	            "Cip".obiekt[#nr].inStartAuto := "Cip".obiekt["Cip".tor[2].pompkaDozowaniaDezynfekantuwLinię].outStartUrządzenie;
	      
	        0:
	            "Cip".obiekt[#nr].Flipaj.in := 0;
	    END_CASE;
	END_REGION
	    
	    REGION ZAWOR ZRZUTOWY DO KANALIZACJI
	    
	    
	        #nr := "Cip".tor[2].zawórZrzutowyDoKanalizacji;
	    CASE "Tor2_program".program.numerKroku OF
	    7100, 7202..7246, 7270,7287,7310, 7320, 7321, 7402, 7403, 7411..7414, 7420, 7431..7435, 7440, 7460:
	    "Cip".obiekt[#nr].procedura := 2;
	   
	    ELSE
	    "Cip".obiekt[#nr].procedura := 0;
	    
	    END_CASE;
	    
	    CASE "Cip".obiekt[#nr].procedura OF
	    2:
	    //wyzwolenie timerków
	    "Cip".obiekt[#nr].SetReset.czasDoSet := 2;
	    "Cip".obiekt[#nr].SetReset.inSet :=
	    "Cip".obiekt["Cip".tor[2].zawórPowrotnyWodyWtórnej].outStartUrządzenie
	    OR "Cip".obiekt["Cip".tor[2].zawórPowrotnyŁugu].outStartUrządzenie
	    OR "Cip".obiekt["Cip".tor[2].zawórPowrotnyKwasu].outStartUrządzenie;
	    
	    "Cip".obiekt[#nr].SetReset.czasDoReset := 2;
	    "Cip".obiekt[#nr].SetReset.inReset :=
	    NOT "Cip".obiekt["Cip".tor[2].zawórPowrotnyWodyWtórnej].outStartUrządzenie
	    AND NOT "Cip".obiekt["Cip".tor[2].zawórPowrotnyŁugu].outStartUrządzenie
	    AND NOT "Cip".obiekt["Cip".tor[2].zawórPowrotnyKwasu].outStartUrządzenie;
	    //załaczanie
	    "Cip".obiekt[#nr].inStartAuto := "Cip".obiekt[#nr].SetReset.wyjście;
	    
	    3:
	    //wyzwolenie timerków
	    "Cip".obiekt[#nr].SetReset.czasDoSet := 2;
	    "Cip".obiekt[#nr].SetReset.inSet :=
	    "Cip".obiekt["Cip".tor[2].zawórBypassPrzygotowaniaStacji].outStartUrządzenie;
	    
	    
	    "Cip".obiekt[#nr].SetReset.czasDoReset := 2;
	    "Cip".obiekt[#nr].SetReset.inReset :=
	    NOT "Cip".obiekt["Cip".tor[2].zawórBypassPrzygotowaniaStacji].outStartUrządzenie;
	    
	    //załaczanie
	    "Cip".obiekt[#nr].inStartAuto := "Cip".obiekt[#nr].SetReset.wyjście;
	    END_CASE;
	    END_REGION
	    
	    REGION ZAWOR WYDAWCZY CIP
	    
	        #nr := "Cip".tor[2].zawórWydawczyCip;
	    CASE "Tor2_program".program.numerKroku OF
	    7210..7290:
	    "Cip".obiekt[#nr].procedura := 1;
	    
	    ELSE
	    "Cip".obiekt[#nr].procedura := 0;
	    
	    END_CASE;
	    
	    CASE "Cip".obiekt[#nr].procedura OF
	    2:
	    //wyzwolenie timerków
	    "Cip".obiekt[#nr].SetReset.czasDoSet := 2;
	    "Cip".obiekt[#nr].SetReset.inSet :=
	    "Cip".obiekt["Cip".tor[2].pompaPodawaniaCip].outStartUrządzenie;
	    
	    "Cip".obiekt[#nr].SetReset.czasDoReset := 2;
	    "Cip".obiekt[#nr].SetReset.inReset :=
	    NOT "Cip".obiekt["Cip".tor[2].pompaPodawaniaCip].outStartUrządzenie;
	    //załaczanie
	    "Cip".obiekt[#nr].inStartAuto := "Cip".obiekt[#nr].SetReset.wyjście;
	    
	    END_CASE;
	    END_REGION
	    
	    REGION ZAWOR BYPASS PRZYGOTOWANIA STACJI
	    
	        #nr := "Cip".tor[2].zawórBypassPrzygotowaniaStacji;
	    CASE "Tor2_program".program.numerKroku OF
	    7210..7290:
	    "Cip".obiekt[#nr].procedura := 2;
	    7320:
	    "Cip".obiekt[#nr].procedura := 3;
	    ELSE
	    "Cip".obiekt[#nr].procedura := 0;
	    
	    END_CASE;
	    CASE "Cip".obiekt[#nr].procedura OF
	    2:
	    //wyzwolenie timerków
	    "Cip".obiekt[#nr].SetReset.czasDoSet := 2;
	    "Cip".obiekt[#nr].SetReset.inSet :=NOT 
	    "Cip".obiekt["Cip".tor[2].zawórWydawczyCip].outStartUrządzenie;
	    
	    "Cip".obiekt[#nr].SetReset.czasDoReset := 2;
	    "Cip".obiekt[#nr].SetReset.inReset :=
	    "Cip".obiekt["Cip".tor[2].zawórWydawczyCip].outStartUrządzenie;
	    //załaczanie
	    "Cip".obiekt[#nr].inStartAuto := "Cip".obiekt[#nr].SetReset.wyjście;
	    3:
	    
	    //załaczanie
	    "Cip".obiekt[#nr].inStartAuto := 1;
	    
	    END_CASE;
	    END_REGION
	    
	    REGION ZAWOR WYDAWCZY WODY WTORNEJ
	    
	        #nr := "Cip".tor[2].zawórWydawczyWodyWtórnej;
	    
	    CASE "Tor2_program".program.numerKroku OF
	    7210,7230:
	    "Cip".obiekt[#nr].procedura := 2;
	    7100:
	    "Cip".obiekt[#nr].procedura := 3;
	    ELSE
	    "Cip".obiekt[#nr].procedura := 0;
	    
	    END_CASE;
	    
	    
	    
	    CASE "Cip".obiekt[#nr].procedura OF
	    2:
	    //wyzwolenie timerków
	    "Cip".obiekt[#nr].SetReset.czasDoSet := 3;
	    "Cip".obiekt[#nr].SetReset.inSet :=
	    "Cip".obiekt["Cip".tor[0].zbiornikWodyWtórnej.czujnikDolnegoPoziomu].hmiPotwWysterowania
	    AND (#aktualnyKrokMycia = 1 OR #aktualnyKrokMycia = 2);
	    
	    "Cip".obiekt[#nr].SetReset.czasDoReset := 10;
	    "Cip".obiekt[#nr].SetReset.inReset :=
	    NOT "Cip".obiekt["Cip".tor[0].zbiornikWodyWtórnej.czujnikDolnegoPoziomu].hmiPotwWysterowania
	    OR (#aktualnyKrokMycia <> 1 AND #aktualnyKrokMycia <> 2);
	    //załaczanie
	    "Cip".obiekt[#nr].inStartAuto := "Cip".obiekt[#nr].SetReset.wyjście;
	    3:
	    //wyzwolenie timerków
	    "Cip".obiekt[#nr].SetReset.czasDoSet := 3;
	    "Cip".obiekt[#nr].SetReset.inSet :=
	    ("Tor2_program".program.numerKroku >= 7401 AND
	    "Tor2_program".program.numerKroku <= 7420);
	    
	    
	    "Cip".obiekt[#nr].SetReset.czasDoReset := 60;
	    "Cip".obiekt[#nr].SetReset.inReset :=
	    NOT ("Tor2_program".program.numerKroku >= 7401 AND
	    "Tor2_program".program.numerKroku <= 7420);
	    
	    //załaczanie
	    "Cip".obiekt[#nr].inStartAuto := "Cip".obiekt[#nr].SetReset.wyjście;
	    
	    END_CASE;
	    END_REGION
	    
	    REGION ZAWÓR POWROTNY WODY WTORNEJ
	    
	        #nr := "Cip".tor[2].zawórPowrotnyWodyWtórnej;
	    CASE "Tor2_program".program.numerKroku OF
	        7250, 7270, 7285, 7287:
	            "Cip".obiekt[#nr].procedura := 2;
	        7402, 7403, 7411, 7414, 7420:
	            "Cip".obiekt[#nr].procedura := 1;
	        ELSE
	            "Cip".obiekt[#nr].procedura := 0;
	            
	    END_CASE;
	    
	    CASE "Cip".obiekt[#nr].procedura OF
	    2:
	    //wyzwolenie timerków
	    "Cip".obiekt[#nr].SetReset.czasDoSet := 1;
	    "Cip".obiekt[#nr].SetReset.inSet :=
	    NOT "Cip".obiekt["Cip".tor[0].zbiornikWodyWtórnej.czujnikGórnegoPoziomu].hmiPotwWysterowania
	    // AND (#aktualnyKrokMycia = 5 OR #aktualnyKrokMycia = 6); // nie wiem czy to było dobrze w Orle 1
	    ;
	    "Cip".obiekt[#nr].SetReset.czasDoReset := 1;
	    "Cip".obiekt[#nr].SetReset.inReset :=
	    "Cip".obiekt["Cip".tor[0].zbiornikWodyWtórnej.czujnikGórnegoPoziomu].hmiPotwWysterowania
	    // OR (#aktualnyKrokMycia <> 5 AND #aktualnyKrokMycia <> 6);
	     ;
	    // ;
	    //załaczanie
	    "Cip".obiekt[#nr].inStartAuto := "Cip".obiekt[#nr].SetReset.wyjście;
	    
	    
	    END_CASE;
	    END_REGION
	    
	    REGION ZAWOR WYDAWCZY ŁUGU
	    
	        #nr := "Cip".tor[2].zawórWydawczyŁugu;
	        CASE "Tor2_program".program.numerKroku OF
	            7240..7243,7411,7412:
	                "Cip".obiekt[#nr].procedura := 2;
	            7100:
	                "Cip".obiekt[#nr].procedura := 3;
	            7320:
	                "Cip".obiekt[#nr].procedura := 4;
	            ELSE
	                "Cip".obiekt[#nr].procedura := 0;
	                
	        END_CASE;
	        
	    CASE "Cip".obiekt[#nr].procedura OF
	    2:
	    //wyzwolenie timerków
	    "Cip".obiekt[#nr].SetReset.czasDoSet := 3;
	    "Cip".obiekt[#nr].SetReset.inSet :=
	    "Cip".obiekt["Cip".tor[0].zbiornikŁugu.czujnikDolnegoPoziomu].hmiPotwWysterowania
	    AND (#aktualnyKrokMycia = 3);
	    
	    "Cip".obiekt[#nr].SetReset.czasDoReset := 10;
	    "Cip".obiekt[#nr].SetReset.inReset :=
	    NOT "Cip".obiekt["Cip".tor[0].zbiornikŁugu.czujnikDolnegoPoziomu].hmiPotwWysterowania
	    OR (#aktualnyKrokMycia <> 3);
	    //załaczanie
	    "Cip".obiekt[#nr].inStartAuto := "Cip".obiekt[#nr].SetReset.wyjście;
	    3:
	    //wyzwolenie timerków
	    "Cip".obiekt[#nr].SetReset.czasDoSet := 3;
	    "Cip".obiekt[#nr].SetReset.inSet :=
	    ("Tor2_program".program.numerKroku >= 7430 AND
	    "Tor2_program".program.numerKroku <= 7440);
	    
	    
	    "Cip".obiekt[#nr].SetReset.czasDoReset := 3;
	    "Cip".obiekt[#nr].SetReset.inReset :=
	    NOT ("Tor2_program".program.numerKroku >= 7430 AND
	    "Tor2_program".program.numerKroku <= 7440);
	    
	    //załaczanie
	    "Cip".obiekt[#nr].inStartAuto := "Cip".obiekt[#nr].SetReset.wyjście;
	    
	    4:
	    //wyzwolenie timerków
	    "Cip".obiekt[#nr].SetReset.czasDoSet := 3;
	    "Cip".obiekt[#nr].SetReset.inSet :=
	    "Cip".obiekt["Cip".tor[0].zbiornikŁugu.czujnikGórnegoPoziomu].hmiPotwWysterowania
	    AND (#aktualnyKrokMycia = 3);
	    
	    
	    
	    "Cip".obiekt[#nr].SetReset.czasDoReset := 3;
	    "Cip".obiekt[#nr].SetReset.inReset :=
	    NOT "Cip".obiekt["Cip".tor[0].zbiornikŁugu.czujnikGórnegoPoziomu].hmiPotwWysterowania
	    OR (#aktualnyKrokMycia <> 3);
	    
	    //załaczanie
	    "Cip".obiekt[#nr].inStartAuto := "Cip".obiekt[#nr].SetReset.wyjście;
	    
	    
	    
	    
	    
	    
	    
	    
	    END_CASE;
	    END_REGION
	    
	    REGION ZAWÓR POWROTNY ŁUGU
	    
	        #nr := "Cip".tor[2].zawórPowrotnyŁugu;
	        CASE "Tor2_program".program.numerKroku OF
	            7431,7432,7434,7435,7440:
	                "Cip".obiekt[#nr].procedura := 1;
	            7242, 7245, 7246, 7321:
	                "Cip".obiekt[#nr].procedura := 2;
	            7100:
	                "Cip".obiekt[#nr].procedura := 3;
	            7243, 7244, 7310, 7320:
	                "Cip".obiekt[#nr].procedura := 4;
	            ELSE
	                "Cip".obiekt[#nr].procedura := 0;
	        END_CASE;
	        
	    CASE "Cip".obiekt[#nr].procedura OF
	    2:
	    //wyzwolenie timerków
	    "Cip".obiekt[#nr].SetReset.czasDoSet := 1;
	    "Cip".obiekt[#nr].SetReset.inSet :=
	    "Cip".obiekt["Cip".tor[2].przewodnośćNaPowrocie].WartośćPomiaru >=
	    "Tor2_RecepturyStacjaMycia".Receptura[#aktualnyNumerReceptury].Krok[#aktualnyKrokMycia].PM[10]
	    AND (#aktualnyKrokMycia = 3)
	    AND NOT "Cip".obiekt["Cip".tor[0].zbiornikŁugu.czujnikGórnegoPoziomu].hmiPotwWysterowania;
	    
	    "Cip".obiekt[#nr].SetReset.czasDoReset := 1;
	    "Cip".obiekt[#nr].SetReset.inReset :=
	    "Cip".obiekt["Cip".tor[2].przewodnośćNaPowrocie].WartośćPomiaru <
	    "Tor2_RecepturyStacjaMycia".Receptura[#aktualnyNumerReceptury].Krok[#aktualnyKrokMycia].PM[10]
	    OR (#aktualnyKrokMycia <> 3)
	    OR "Cip".obiekt["Cip".tor[0].zbiornikŁugu.czujnikGórnegoPoziomu].hmiPotwWysterowania;
	    //załaczanie
	    "Cip".obiekt[#nr].inStartAuto := "Cip".obiekt[#nr].SetReset.wyjście;
	    3:
	    //wyzwolenie timerków
	    "Cip".obiekt[#nr].SetReset.czasDoSet := 3;
	    "Cip".obiekt[#nr].SetReset.inSet :=
	    "Cip".obiekt["Cip".tor[2].zawórWydawczyŁugu].inStartAuto
	    AND ("Tor2_program".program.numerKroku > 7400
	    AND "Tor2_program".program.numerKroku < 7470);
	    
	    
	    "Cip".obiekt[#nr].SetReset.czasDoReset := 3;
	    "Cip".obiekt[#nr].SetReset.inReset :=
	    NOT "Cip".obiekt["Cip".tor[2].zawórWydawczyŁugu].inStartAuto
	    OR ("Tor2_program".program.numerKroku < 7400
	    OR "Tor2_program".program.numerKroku > 7470);
	    
	    //załaczanie
	    "Cip".obiekt[#nr].inStartAuto := "Cip".obiekt[#nr].SetReset.wyjście;
	    
	    4:
	    //wyzwolenie timerków
	    "Cip".obiekt[#nr].SetReset.czasDoSet := 3;
	    "Cip".obiekt[#nr].SetReset.inSet :=
	    (#aktualnyKrokMycia = 3);
	    
	    "Cip".obiekt[#nr].SetReset.czasDoReset := 10;
	    "Cip".obiekt[#nr].SetReset.inReset :=
	    (#aktualnyKrokMycia <> 3);
	    //załaczanie
	    "Cip".obiekt[#nr].inStartAuto := "Cip".obiekt[#nr].SetReset.wyjście;
	    END_CASE;
	    
	    END_REGION
	    
	    REGION ZAWÓR WYDAWCZY KWASU
	        
	        #nr := "Cip".tor[2].zawórWydawczyKwasu;
	        CASE "Tor2_program".program.numerKroku OF
	            7240..7243, 7411, 7412, 7434, 7435:
	                "Cip".obiekt[#nr].procedura := 2;
	            7100:
	                "Cip".obiekt[#nr].procedura := 3;
	            7320:
	                "Cip".obiekt[#nr].procedura := 4;
	            ELSE
	                "Cip".obiekt[#nr].procedura := 0;
	                
	        END_CASE;
	        
	        CASE "Cip".obiekt[#nr].procedura OF
	            2:
	                //wyzwolenie timerków
	                "Cip".obiekt[#nr].SetReset.czasDoSet := 3;
	                "Cip".obiekt[#nr].SetReset.inSet :=
	                "Cip".obiekt["Cip".tor[0].zbiornikKwasu.czujnikDolnegoPoziomu].hmiPotwWysterowania
	                AND (#aktualnyKrokMycia = 4);
	                
	                "Cip".obiekt[#nr].SetReset.czasDoReset := 10;
	                "Cip".obiekt[#nr].SetReset.inReset :=
	                NOT "Cip".obiekt["Cip".tor[0].zbiornikKwasu.czujnikDolnegoPoziomu].hmiPotwWysterowania
	                OR (#aktualnyKrokMycia <> 4);
	                
	                //załaczanie
	                "Cip".obiekt[#nr].inStartAuto := "Cip".obiekt[#nr].SetReset.wyjście;
	            3:
	                //wyzwolenie timerków
	                "Cip".obiekt[#nr].SetReset.czasDoSet := 3;
	                "Cip".obiekt[#nr].SetReset.inSet :=
	                ("Tor2_program".program.numerKroku >= 7450 AND
	                "Tor2_program".program.numerKroku <= 7470);
	                
	                
	                "Cip".obiekt[#nr].SetReset.czasDoReset := 3;
	                "Cip".obiekt[#nr].SetReset.inReset :=
	                NOT ("Tor2_program".program.numerKroku >= 7450 AND
	                "Tor2_program".program.numerKroku <= 7470);
	                
	                //załaczanie
	                "Cip".obiekt[#nr].inStartAuto := "Cip".obiekt[#nr].SetReset.wyjście;
	                
	                
	            4:
	                //wyzwolenie timerków
	                "Cip".obiekt[#nr].SetReset.czasDoSet := 3;
	                "Cip".obiekt[#nr].SetReset.inSet :=
	                "Cip".obiekt["Cip".tor[0].zbiornikKwasu.czujnikGórnegoPoziomu].hmiPotwWysterowania
	                AND (#aktualnyKrokMycia = 4);
	                
	                
	                
	                "Cip".obiekt[#nr].SetReset.czasDoReset := 3;
	                "Cip".obiekt[#nr].SetReset.inReset :=
	                NOT "Cip".obiekt["Cip".tor[0].zbiornikKwasu.czujnikGórnegoPoziomu].hmiPotwWysterowania
	                OR (#aktualnyKrokMycia <> 4);
	                
	                //załaczanie
	                "Cip".obiekt[#nr].inStartAuto := "Cip".obiekt[#nr].SetReset.wyjście;
	                
	        END_CASE;
	    END_REGION
	    
	    REGION ZAWÓR POWROTNY KWASU
	        
	        #nr := "Cip".tor[2].zawórPowrotnyKwasu;
	        
	        CASE "Tor2_program".program.numerKroku OF
	            7460:
	                "Cip".obiekt[#nr].procedura := 1;
	            7242, 7245, 7246, 7321:
	                "Cip".obiekt[#nr].procedura := 2;
	            7100:
	                "Cip".obiekt[#nr].procedura := 3;
	            7243, 7244, 7310, 7320:
	                "Cip".obiekt[#nr].procedura := 4;
	            ELSE
	                "Cip".obiekt[#nr].procedura := 0;
	        END_CASE;
	        
	        CASE "Cip".obiekt[#nr].procedura OF
	            2:
	                //wyzwolenie timerków
	                "Cip".obiekt[#nr].SetReset.czasDoSet := 1;
	                "Cip".obiekt[#nr].SetReset.inSet :=
	                "Cip".obiekt["Cip".tor[2].przewodnośćNaPowrocie].WartośćPomiaru >=
	                "Tor2_RecepturyStacjaMycia".Receptura[#aktualnyNumerReceptury].Krok[#aktualnyKrokMycia].PM[10]
	                AND (#aktualnyKrokMycia = 4)
	                AND NOT "Cip".obiekt["Cip".tor[0].zbiornikKwasu.czujnikGórnegoPoziomu].hmiPotwWysterowania;
	                
	                "Cip".obiekt[#nr].SetReset.czasDoReset := 1;
	                "Cip".obiekt[#nr].SetReset.inReset :=
	                "Cip".obiekt["Cip".tor[2].przewodnośćNaPowrocie].WartośćPomiaru <
	                "Tor2_RecepturyStacjaMycia".Receptura[#aktualnyNumerReceptury].Krok[#aktualnyKrokMycia].PM[10]
	                OR (#aktualnyKrokMycia <> 4)
	                OR "Cip".obiekt["Cip".tor[0].zbiornikKwasu.czujnikGórnegoPoziomu].hmiPotwWysterowania;
	                //załaczanie
	                "Cip".obiekt[#nr].inStartAuto := "Cip".obiekt[#nr].SetReset.wyjście;
	            3:
	                //wyzwolenie timerków
	                "Cip".obiekt[#nr].SetReset.czasDoSet := 3;
	                "Cip".obiekt[#nr].SetReset.inSet :=
	                "Cip".obiekt["Cip".tor[2].zawórWydawczyKwasu].inStartAuto AND
	                ("Tor2_program".program.numerKroku >= 7400 AND
	                "Tor2_program".program.numerKroku <= 7470);
	                ;
	                
	                
	                "Cip".obiekt[#nr].SetReset.czasDoReset := 3;
	                "Cip".obiekt[#nr].SetReset.inReset :=
	                NOT "Cip".obiekt["Cip".tor[2].zawórWydawczyKwasu].inStartAuto
	                OR ("Tor2_program".program.numerKroku < 7400 OR
	                "Tor2_program".program.numerKroku > 7470);
	                ;
	                
	                //załaczanie
	                "Cip".obiekt[#nr].inStartAuto := "Cip".obiekt[#nr].SetReset.wyjście;
	            4:
	                //wyzwolenie timerków
	                "Cip".obiekt[#nr].SetReset.czasDoSet := 3;
	                "Cip".obiekt[#nr].SetReset.inSet := (#aktualnyKrokMycia = 4);
	                
	                "Cip".obiekt[#nr].SetReset.czasDoReset := 10;
	                "Cip".obiekt[#nr].SetReset.inReset := (#aktualnyKrokMycia <> 4);
	                
	                //załaczanie
	                "Cip".obiekt[#nr].inStartAuto := "Cip".obiekt[#nr].SetReset.wyjście;
	        END_CASE;
	    END_REGION
	    
	    REGION ZAWÓR WYDAWCZY WODY CZYSTEJ
	    
	        #nr := "Cip".tor[2].zawórWydawczyWodyCzystej;
	        
	        CASE "Tor2_program".program.numerKroku OF
	            7220..7230, 7411, 7412:
	                "Cip".obiekt[#nr].procedura := 2;
	            7244..7270, 7321, 7402, 7403, 7414, 7420, 7431, 7432, 7440, 7460:
	                "Cip".obiekt[#nr].procedura := 3;
	            7242, 7243:
	                "Cip".obiekt[#nr].procedura := 4;
	            7310, 7320:
	                "Cip".obiekt[#nr].procedura := 5;
	            7281..7291:
	                "Cip".obiekt[#nr].procedura := 6;
	            ELSE
	                "Cip".obiekt[#nr].procedura := 0;
	                
	        END_CASE;
	        
	        
	    CASE "Cip".obiekt[#nr].procedura OF
	    2:
	    //wyzwolenie timerków
	    "Cip".obiekt[#nr].SetReset.czasDoSet := 3;
	    "Cip".obiekt[#nr].SetReset.inSet :=
	    "Cip".obiekt["Cip".tor[0].zbiornikwodyCzystej.czujnikDolnegoPoziomu].hmiPotwWysterowania
	    AND NOT "Cip".obiekt["Cip".tor[0].zbiornikWodyWtórnej.czujnikDolnegoPoziomu].hmiPotwWysterowania;
	    
	    "Cip".obiekt[#nr].SetReset.czasDoReset := 10;
	    "Cip".obiekt[#nr].SetReset.inReset :=
	    NOT "Cip".obiekt["Cip".tor[0].zbiornikwodyCzystej.czujnikDolnegoPoziomu].hmiPotwWysterowania
	    OR "Cip".obiekt["Cip".tor[0].zbiornikWodyWtórnej.czujnikDolnegoPoziomu].hmiPotwWysterowania;
	    //załaczanie
	    "Cip".obiekt[#nr].inStartAuto := "Cip".obiekt[#nr].SetReset.wyjście;
	    3:
	    //wyzwolenie timerków
	    "Cip".obiekt[#nr].SetReset.czasDoSet := 3;
	    "Cip".obiekt[#nr].SetReset.inSet :=
	    "Cip".obiekt["Cip".tor[0].zbiornikwodyCzystej.czujnikDolnegoPoziomu].hmiPotwWysterowania;
	    
	    
	    "Cip".obiekt[#nr].SetReset.czasDoReset := 3;
	    "Cip".obiekt[#nr].SetReset.inReset :=
	    NOT "Cip".obiekt["Cip".tor[0].zbiornikwodyCzystej.czujnikDolnegoPoziomu].hmiPotwWysterowania;
	    
	    //załaczanie
	    "Cip".obiekt[#nr].inStartAuto := "Cip".obiekt[#nr].SetReset.wyjście;
	    
	    4:
	    //wyzwolenie timerków
	    "Cip".obiekt[#nr].SetReset.czasDoSet := 1;
	    "Cip".obiekt[#nr].SetReset.inSet :=
	    (NOT "Cip".obiekt["Cip".tor[0].zbiornikŁugu.czujnikDolnegoPoziomu].hmiPotwWysterowania AND #aktualnyKrokMycia = 3)
	    OR (NOT "Cip".obiekt["Cip".tor[0].zbiornikKwasu.czujnikDolnegoPoziomu].hmiPotwWysterowania AND #aktualnyKrokMycia = 4);
	    
	    
	    "Cip".obiekt[#nr].SetReset.czasDoReset := 5;
	    "Cip".obiekt[#nr].SetReset.inReset :=
	    ("Cip".obiekt["Cip".tor[0].zbiornikŁugu.czujnikDolnegoPoziomu].hmiPotwWysterowania AND #aktualnyKrokMycia = 3)
	    OR ("Cip".obiekt["Cip".tor[0].zbiornikKwasu.czujnikDolnegoPoziomu].hmiPotwWysterowania AND #aktualnyKrokMycia = 4);
	    //załaczanie
	    "Cip".obiekt[#nr].inStartAuto := "Cip".obiekt[#nr].SetReset.wyjście;
	    
	    5:
	    //wyzwolenie timerków
	    "Cip".obiekt[#nr].SetReset.czasDoSet := 1;
	    "Cip".obiekt[#nr].SetReset.inSet :=
	    (NOT "Cip".obiekt["Cip".tor[0].zbiornikŁugu.czujnikGórnegoPoziomu].hmiPotwWysterowania AND #aktualnyKrokMycia = 3)
	    OR (NOT "Cip".obiekt["Cip".tor[0].zbiornikKwasu.czujnikGórnegoPoziomu].hmiPotwWysterowania AND #aktualnyKrokMycia = 4);
	    
	    
	    "Cip".obiekt[#nr].SetReset.czasDoReset := 2;
	    "Cip".obiekt[#nr].SetReset.inReset :=
	    ("Cip".obiekt["Cip".tor[0].zbiornikŁugu.czujnikGórnegoPoziomu].hmiPotwWysterowania AND #aktualnyKrokMycia = 3)
	    OR ("Cip".obiekt["Cip".tor[0].zbiornikKwasu.czujnikGórnegoPoziomu].hmiPotwWysterowania AND #aktualnyKrokMycia = 4);
	    //załaczanie
	    "Cip".obiekt[#nr].inStartAuto := "Cip".obiekt[#nr].SetReset.wyjście;
	6:
	    //wyzwolenie timerków
	    "Cip".obiekt[#nr].SetReset.czasDoSet :=1;
	    "Cip".obiekt[#nr].SetReset.inSet :=
	    NOT ("Cip".obiekt["Cip".tor[2].zawórWydawczyDezynfekantu].hmiPotwWysterowania);
	    
	    
	    "Cip".obiekt[#nr].SetReset.czasDoReset := 2;
	    "Cip".obiekt[#nr].SetReset.inReset :=
	    ("Cip".obiekt["Cip".tor[2].zawórWydawczyDezynfekantu].hmiPotwWysterowania);;
	    //załaczanie
	    "Cip".obiekt[#nr].inStartAuto := "Cip".obiekt[#nr].SetReset.wyjście;
	    
	    END_CASE;
	    END_REGION
	    
	    REGION zawór wydawczy dezynfekantu
	        
	        #nr := "Cip".tor[2].zawórWydawczyDezynfekantu;
	        CASE "Tor2_program".program.numerKroku OF
	            7282..7284:
	                "Cip".obiekt[#nr].procedura := 2;
	                
	            ELSE
	                "Cip".obiekt[#nr].procedura := 0;
	                
	        END_CASE;
	        
	        CASE "Cip".obiekt[#nr].procedura OF
	            2:
	                //wyzwolenie timerków
	                "Cip".obiekt[#nr].SetReset.czasDoSet := 2;
	                "Cip".obiekt[#nr].SetReset.inSet :=
	                "Cip".obiekt["Cip".tor[2].zbiornikDezynfekantu.poziomAnalogowy].WartośćPomiaru > 10.0;
	                
	                "Cip".obiekt[#nr].SetReset.czasDoReset := 2;
	                "Cip".obiekt[#nr].SetReset.inReset :=
	                "Cip".obiekt["Cip".tor[2].zbiornikDezynfekantu.poziomAnalogowy].WartośćPomiaru < 0.01;
	                ;
	                //załaczanie
	                "Cip".obiekt[#nr].inStartAuto := "Cip".obiekt[#nr].SetReset.wyjście;
	                
	        END_CASE;
	    END_REGION
	    
	    REGION zawór powrotny dezynfekantu
	        
	        #nr := "Cip".tor[2].zawórPowrotnyDezynfekantu;
	        CASE "Tor2_program".program.numerKroku OF
	            7281..7283:
	                "Cip".obiekt[#nr].procedura :=2;
	                
	            ELSE
	                "Cip".obiekt[#nr].procedura := 0;
	                
	        END_CASE;
	        
	        CASE "Cip".obiekt[#nr].procedura OF
	            2:
	                //wyzwolenie timerków
	                "Cip".obiekt[#nr].SetReset.czasDoSet := 5;
	                "Cip".obiekt[#nr].SetReset.inSet :=
	                NOT  "Cip".obiekt["Cip".tor[2].zbiornikDezynfekantu.czujnikGórnegoPoziomu].hmiPotwWysterowania ;
	                
	                "Cip".obiekt[#nr].SetReset.czasDoReset := 0;
	                "Cip".obiekt[#nr].SetReset.inReset :=
	                "Cip".obiekt["Cip".tor[2].zbiornikDezynfekantu.czujnikGórnegoPoziomu].hmiPotwWysterowania;
	                ;
	                //załaczanie
	                "Cip".obiekt[#nr].inStartAuto := "Cip".obiekt[#nr].SetReset.wyjście;
	                
	        END_CASE;
	    END_REGION
	    
	    REGION zawór stopowy dezynfekantu
	        
	        #nr := "Cip".tor[2].zawórStopowyPowrotuDezynfekantu;
	        CASE "Tor2_program".program.numerKroku OF
	            7281..7283:
	                "Cip".obiekt[#nr].procedura := 2;
	                
	            ELSE
	                "Cip".obiekt[#nr].procedura := 0;
	                
	        END_CASE;
	        
	        CASE "Cip".obiekt[#nr].procedura OF
	            2:
	                //wyzwolenie timerków
	                "Cip".obiekt[#nr].SetReset.czasDoSet := 0;
	                "Cip".obiekt[#nr].SetReset.inSet :=
	                "Cip".obiekt["Cip".tor[2].zawórPowrotnyDezynfekantu].hmiPotwWysterowania;
	                
	                "Cip".obiekt[#nr].SetReset.czasDoReset := 0;
	                "Cip".obiekt[#nr].SetReset.inReset :=
	                NOT "Cip".obiekt["Cip".tor[2].zawórPowrotnyDezynfekantu].hmiPotwWysterowania;
	                ;
	                //załaczanie
	                "Cip".obiekt[#nr].inStartAuto := "Cip".obiekt[#nr].SetReset.wyjście;
	                
	        END_CASE;
	    END_REGION
	    
	    REGION ZAWÓR PAROWY REGULACYJNY
	    
	        #nr := "Cip".tor[2].zawórParowyRegulacyjny;
	        
	    CASE "Tor2_program".program.numerKroku OF
	    7220, 7250, 7403, 7414, 7432:
	    "Cip".obiekt[#nr].procedura := 2;
	    7242..7246, 7320, 7321, 7411, 7412, 7434, 7435:
	    "Cip".obiekt[#nr].procedura := 3;
	    
	    ELSE
	    "Cip".obiekt[#nr].procedura := 0;
	    
	    END_CASE;
	    
	    
	    CASE "Cip".obiekt[#nr].procedura OF
	    2:
	    //wyzwolenie timerków
	    "Cip".obiekt[#nr].SetReset.czasDoSet := 2;
	    "Cip".obiekt[#nr].SetReset.inSet := "Cip".obiekt["Cip".tor[2].zawórParowyOdcinający].outStartUrządzenie;
	    
	    "Cip".obiekt[#nr].SetReset.czasDoReset := 2;
	    "Cip".obiekt[#nr].SetReset.inReset := NOT "Cip".obiekt["Cip".tor[2].zawórParowyOdcinający].outStartUrządzenie;
	    
	    
	    //załaczanie
	    "Cip".obiekt[#nr].inStartAuto := "Cip".obiekt[#nr].SetReset.wyjście;
	    
	    //wysterowanie
	    "Cip".obiekt[#nr].inZadaneWysterowanieAuto :=  //pid_out wypełniamy w wywołaniu pida z out pida
	    LIMIT(IN := "Cip".obiekt[#nr].pid_Out, MN := 0.0, MX := 100.0);//pid_out ;
	    
	    ////PID
	    "Cip".obiekt[#nr].pid_SP :=
	    "Tor2_RecepturyStacjaMycia".Receptura[#aktualnyNumerReceptury].Krok[#aktualnyKrokMycia].PM[14];
	    "Cip".obiekt[#nr].pid_PV := "Cip".obiekt["Cip".tor[2].temperaturaZaWymiennikiem].WartośćPomiaru;
	    3:
	    //wyzwolenie timerków
	    "Cip".obiekt[#nr].SetReset.czasDoSet := 2;
	    "Cip".obiekt[#nr].SetReset.inSet := "Cip".obiekt["Cip".tor[2].zawórParowyOdcinający].outStartUrządzenie;
	    
	    "Cip".obiekt[#nr].SetReset.czasDoReset := 2;
	    "Cip".obiekt[#nr].SetReset.inReset := NOT "Cip".obiekt["Cip".tor[2].zawórParowyOdcinający].outStartUrządzenie;
	    
	    
	    //załaczanie
	    "Cip".obiekt[#nr].inStartAuto := "Cip".obiekt[#nr].SetReset.wyjście;
	    
	    //wysterowanie
	    "Cip".obiekt[#nr].inZadaneWysterowanieAuto :=  //pid_out wypełniamy w wywołaniu pida z out pida
	    LIMIT(IN := "Cip".obiekt[#nr].pid_Out, MN := 0.0, MX := 100.0);//pid_out ;
	    
	    ////PID
	    "Cip".obiekt[#nr].pid_SP :=
	    "Tor2_RecepturyStacjaMycia".Receptura[#aktualnyNumerReceptury].Krok[#aktualnyKrokMycia].PM[13];
	    "Cip".obiekt[#nr].pid_PV := "Cip".obiekt["Cip".tor[2].temperaturaZaWymiennikiem].WartośćPomiaru;
	    
	    0:
	    ;
	    
	    // resetowanie całkującej części regulatora aby nie przejebać temperatury
	    // "PID_Compact23".IntegralResetMode := 3;
	    // "PID_Compact23".OverwriteInitialOutputValue := "F1.SP"."203"- 1.0;
	    // "PID_Compact23".Reset := "F1".obiekt["F100LT01"].WartośćPomiaru > 70.0;
	    // := LIMIT(IN := "APA".obiekt["PID123"].outWysterowanieUrządzenia,
	    // MN := 0.0, MX := "APA".obiekt["H101TT01"].WartośćPomiaru + "H1.STP"."214");
	    
	    END_CASE;
	    
	    IF "Cip".obiekt[#nr].procedura > 0 THEN
	    
	    IF "Cip".obiekt[#nr].inStartAuto = 0 THEN
	    "Cip".obiekt[#nr].inZadaneWysterowanieAuto := 0.0;
	    "Cip".obiekt[#nr].pid_SP := 0.0;
	    END_IF;
	    END_IF;
	    
	    
	    "PID.zawórRegulacyjnyParyTor1"(Setpoint := "Cip".obiekt[#nr].pid_SP,
	                           Input := "Cip".obiekt[#nr].pid_PV,
	                           Reset := "Cip".obiekt[#nr].hmiResetAwaria,
	                           Output => "Cip".obiekt[#nr].pid_Out);
	    "PID.zawórRegulacyjnyParyTor1".Retain.CtrlParams.Gain := 1.0;
	    "PID.zawórRegulacyjnyParyTor1".Retain.CtrlParams.Ti := "Cip".obiekt[#nr].pid_I;
	    "PID.zawórRegulacyjnyParyTor1".Retain.CtrlParams.Td := "Cip".obiekt[#nr].pid_D;
	END_REGION
	
	    REGION ZAWOR PAROWY ODCINAJACY
	        
	        #nr := "Cip".tor[2].zawórParowyOdcinający;
	        CASE "Tor2_program".program.numerKroku OF
	            7220, 7240, 7242,7243, 7246, 7250, 7320, 7321, 7403, 7411, 7412, 7414, 7432, 7434, 7435:
	                "Cip".obiekt[#nr].procedura := 2;
	                
	            ELSE
	                "Cip".obiekt[#nr].procedura := 0;
	                
	        END_CASE;
	        
	        CASE "Cip".obiekt[#nr].procedura OF
	            2:
	                //wyzwolenie timerków
	                "Cip".obiekt[#nr].SetReset.czasDoSet := 2;
	                "Cip".obiekt[#nr].SetReset.inSet :=
	                "Cip".obiekt["Cip".tor[2].pompaPodawaniaCip].hmiPotwWysterowania
	                AND "Cip".obiekt["Cip".tor[2].temperaturaZaWymiennikiem].WartośćPomiaru < 90;
	                
	                "Cip".obiekt[#nr].SetReset.czasDoReset := 2;
	                "Cip".obiekt[#nr].SetReset.inReset :=
	                NOT "Cip".obiekt["Cip".tor[2].pompaPodawaniaCip].hmiPotwWysterowania
	                OR "Cip".obiekt["Cip".tor[2].temperaturaZaWymiennikiem].WartośćPomiaru >= 95;
	                //załaczanie
	                "Cip".obiekt[#nr].inStartAuto := "Cip".obiekt[#nr].SetReset.wyjście;
	        END_CASE;
	    END_REGION
	            
END_FUNCTION

FUNCTION "Tor2.procedury_sygnałów" : Void
{ S7_Optimized_Access := 'TRUE' }
VERSION : 0.1
   VAR_TEMP 
      x : Int;
      y : Int;
      numerProcedury : Int;
      indexKroku : Int;
      numerObiektu : Int;
      aktualnyNumerReceptury : Int;
      aktualnyKrokMycia : Int;
   END_VAR

   VAR CONSTANT 
      "1" : Int := 1;
      CIP2 : Int := 2;
      CIP3 : Int := 3;
      TANK_CIP : Int := 4;
      READY1 : Int := 5;
      READY2 : Int := 6;
      READY3 : Int := 7;
      CONF1 : Int := 8;
      CONF2 : Int := 9;
      ERR : Int := 10;
      PULLOUT1 : Int := 11;
      PULLOUT2 : Int := 12;
      PULLOUT3 : Int := 13;
      WATER1 : Int := 14;
      WATER2 : Int := 15;
      WATER3 : Int := 16;
      OUT1 : Int := 17;
      OUT2 : Int := 18;
      OUT3 : Int := 19;
      CONNECT1 : Int := 20;
      CONNECT2 : Int := 21;
      CONNECT3 : Int := 22;
      WHEY : Int := 23;
      AG : Int := 24;
      PUMP : Int := 25;
      FLIP : Int := 26;
      S1_RUNNING : Int := 27;
      S1_FEED : Int := 28;
      S1_START : Int := 29;
      S1_REMOTE : Int := 30;
      S1_RINSING : Int := 31;
      S1_ERR : Int := 32;
      S1_OUT : Int := 33;
   END_VAR


BEGIN
	
	// //=============================================================================
	// // Mlekomat Sp. z o.o.// (c)Copyright (2019)
	// //-----------------------------------------------------------------------------
	// // Biblioteka: Orzeł-Piotr Kowalski
	// // Testowano za pomocą: PLCSIM Advanced v.2.0 sp1
	// // Engineering: TIA Portal 15.1
	// // Ograniczenia: (typy bloków OB, itp.)
	// // Wymagania: (sprzęt, pamięć, itp.)
	// // Funkcjonalność:  Odczytanie z tablicy  "F1.sygnały.1_99.krok" numeru procedury
	// // dla każdego sygnału "Sygnały".F[1]....   i zastosowanie oewj procedury - zgodnie
	// // z dokumentem FD od technologa
	// //----------------------------------------------------------------------------
	// // Zmiany w logu:
	// // Wersja Data Autor Data wprowadzenia zmian
	// // 01.00.00 15.03.2019 Piotr Kowalski//
	// //=============================================================================
	
	// //program zawiera procedury dla sygnałów dla procedur o numerze >1  (procedura 0 i 1 jest obsługiwana w programie FB_obsługa sygnałów)
	// //procedury wyzwalane  z progrmu TablicaProcedór dla kolejnych kroków  "F1".obiekt["F100CP01"].procedura: = 2
	// //wyzwolenie procedury zero  automatycznie  wyłącza sygnał
	// //procedura:=1   wyzwala sygnał SET -- obsługiwana jest w programie FB obsłóga sygnałów
	// //
	// //
	// //open ctrl+shift+(*)Numeric
	// //close ctrl+shift+(/)Numeric
	// //
	
	// #aktualnyNumerReceptury := "CIP1_RecepturyStacjaMycia".numerUżywanejReceptury;
	// #aktualnyKrokMycia := "CIP1_RecepturyStacjaMycia".numerKrokuMycia;
	
	
	
	
	
	
	// CASE "CIP1_sygnały".sygnał[#"1"].procedura OF
	        
	//     2:
	//         IF "CIP1_RecepturyStacjaMycia".Receptura[#aktualnyNumerReceptury].Krok[#aktualnyKrokMycia].PM[21] = 1 THEN
	//             IF
	//                 ("CIP1_RecepturyStacjaMycia".Receptura[#aktualnyNumerReceptury].Krok[#aktualnyKrokMycia].PM[24] = 2101
	//                 AND "SIG".SIG[2101]=1)
	//                 OR ("CIP1_RecepturyStacjaMycia".Receptura[#aktualnyNumerReceptury].Krok[#aktualnyKrokMycia].PM[24] = 2102
	//                 AND "SIG".SIG[2102]=1)
	//                 OR ("CIP1_RecepturyStacjaMycia".Receptura[#aktualnyNumerReceptury].Krok[#aktualnyKrokMycia].PM[24] = 3101
	//                 AND "SIG".SIG[3101]=1)
	//                 OR ("CIP1_RecepturyStacjaMycia".Receptura[#aktualnyNumerReceptury].Krok[#aktualnyKrokMycia].PM[24] = 3102
	//                 AND "SIG".SIG[3102]=1)
	//                 OR ("CIP1_RecepturyStacjaMycia".Receptura[#aktualnyNumerReceptury].Krok[#aktualnyKrokMycia].PM[24] = 9401
	//                 AND "SIG".SIG[9401]=1)
	//                 OR ("CIP1_RecepturyStacjaMycia".Receptura[#aktualnyNumerReceptury].Krok[#aktualnyKrokMycia].PM[24] = 9501
	//                 AND "SIG".SIG[9501]=1)
	//                 OR ("CIP1_RecepturyStacjaMycia".Receptura[#aktualnyNumerReceptury].Krok[#aktualnyKrokMycia].PM[24] = 4101
	//                 AND "SIG".SIG[4101]=1)
	//             THEN
	//                 "CIP1_sygnały".sygnał[#"1"].inStart := 1;
	//             END_IF;
	//             ;
	//         END_IF;
	//     0:
	//         "CIP1_sygnały".sygnał[#"1"].inStart := 0;
	        
	// END_CASE;
	// "SIG".SIG[7101] := BOOL_TO_INT("CIP1_sygnały".sygnał[#"1"].inStart);
	
	// CASE "CIP1_sygnały".sygnał[#OUT1].procedura OF
	        
	//     2:
	        
	      
	//         "CIP1_sygnały".sygnał[#OUT1].inStart := "CIP1_obiekty".obiekt["C101AV13"].outStartUrządzenie;
	    
	//         ;
	//     0:
	//         "CIP1_sygnały".sygnał[#OUT1].inStart := 0;
	        
	// END_CASE;
	// "SIG".SIG[7120] := BOOL_TO_INT("CIP1_sygnały".sygnał[#OUT1].inStart);
	
	
	// CASE "CIP1_sygnały".sygnał[#AG].procedura OF
	        
	//     2:
	//         "Flipaj_cip1_sygnał_AG"(ile_petli := 999,
	//                                 czas_ON   := 100,
	//                                 czas_OFF  := 600);
	        
	        
	//         IF "CIP1_RecepturyStacjaMycia".Receptura[#aktualnyNumerReceptury].Krok[#aktualnyKrokMycia].PM[23]=1 THEN
	//             "Flipaj_cip1_sygnał_AG".in := 1;
	//             "CIP1_sygnały".sygnał[#AG].inStart := "Flipaj_cip1_sygnał_AG".Q;
	//         ELSE
	//             "Flipaj_cip1_sygnał_AG".in := 0;
	//         END_IF;
	//     0:
	//         "Flipaj_cip1_sygnał_AG".in := 0;
	//         "CIP1_sygnały".sygnał[#AG].inStart := 0;
	// END_CASE;
	// "SIG".SIG[7127] := BOOL_TO_INT("CIP1_sygnały".sygnał[#AG].inStart);
	
	
	// CASE "CIP1_sygnały".sygnał[#FLIP].procedura OF
	        
	//     2:
	//         "Flipaj_cip1_sygnał_FLIP"(ile_petli := 999,
	//                                 czas_ON   := 300,
	//                                 czas_OFF  := 600);
	        
	        
	//       // IF "CIP1_RecepturyStacjaMycia".Receptura[#aktualnyNumerReceptury].Krok[#aktualnyKrokMycia].PM[23] = 1
	//           IF 1=1
	//       THEN
	//             "Flipaj_cip1_sygnał_FLIP".in := 1;
	//             "CIP1_sygnały".sygnał[#FLIP].inStart := "Flipaj_cip1_sygnał_FLIP".Q;
	//         ELSE
	//             "Flipaj_cip1_sygnał_FLIP".in := 0;
	//         END_IF;
	//     0:
	     
	//         "CIP1_sygnały".sygnał[#FLIP].inStart := 0;
	//         "Flipaj_cip1_sygnał_FLIP"(in:=0,
	//                                   ile_petli := 999,
	//                                   czas_ON := 300,
	//                                   czas_OFF := 600);
	// END_CASE;
	// "SIG".SIG[7128] := BOOL_TO_INT("CIP1_sygnały".sygnał[#FLIP].inStart);
	
	
	// CASE "CIP1_sygnały".sygnał[#PUMP].procedura OF
	        
	//     2:
	        
	        
	//         IF "CIP1_RecepturyStacjaMycia".Receptura[#aktualnyNumerReceptury].Krok[#aktualnyKrokMycia].PM[23] = 1
	//             AND "licznik_1" < "CIP1_RecepturyStacjaMycia".Receptura[#aktualnyNumerReceptury].Krok[#aktualnyKrokMycia].PM[9] * 10
	//         THEN
	//             "licznik_1" := "licznik_1" + 1;
	//             IF "licznik_1" >= "CIP1_RecepturyStacjaMycia".Receptura[#aktualnyNumerReceptury].Krok[#aktualnyKrokMycia].PM[9] * 10
	//             THEN
	//                 "CIP1_sygnały".sygnał[#PUMP].inStart := 1;
	//             END_IF;
	            
	//         END_IF;
	//     0:
	//         "CIP1_sygnały".sygnał[#PUMP].inStart := 0;
	//         "licznik_1" := 0;
	// END_CASE;
	// "SIG".SIG[7129] := BOOL_TO_INT("CIP1_sygnały".sygnał[#PUMP].inStart);
	
	
	
	// IF "CIP1_hmi".button.bPauza.set THEN
	//     "SIG".SIG[7127] := 0;
	//     "SIG".SIG[7128] := 0;
	//     "SIG".SIG[7129] := 0;
	// END_IF;
	
	
	// "SIG".SIG[7161] := "CIP1_program".program.numerKroku;
	
	// //s1.rinsing
	// IF "CIP1_program".program.numerKroku = 7210
	//     OR "CIP1_program".program.numerKroku = 7220
	//     OR "CIP1_program".program.numerKroku = 7250
	//     OR "CIP1_program".program.numerKroku = 7270
	//     OR "CIP1_program".program.numerKroku = 7282
	    
	// THEN
	//     "SIG".SIG[7134] := 1;
	// ELSE
	//     "SIG".SIG[7134] := 0;
	// END_IF;
	// //s1.out
	// IF ("CIP1_program".program.numerKroku >= 7240
	//     AND "CIP1_program".program.numerKroku <= 7246)
	//     OR "CIP1_program".program.numerKroku = 7280
	//     OR "CIP1_program".program.numerKroku = 7281
	    
	    
	// THEN
	//     "SIG".SIG[7136] := 1;
	// ELSE
	//     "SIG".SIG[7136] := 0;
	// END_IF;
	    
	
	
	
	
	
	
	
	
END_FUNCTION

FUNCTION "Tor0.aMAIN" : Void
{ S7_Optimized_Access := 'TRUE' }
VERSION : 0.1

BEGIN
	"Tor0.procedury_obiektów"();
	
	
	
	
	
	
	
	// //milisimensy na procenty Tor1
	// "ms_na_procenty"(inWartośćMierzona        := "CIP1_obiekty".obiekt["C101CT11"].WartośćPomiaru,
	//                  inJednostkaAlkaliczna    := "ms_na_procenty_DB".inJednostkaAlkaliczna,
	//                  inJednostkaKwaśna        := "ms_na_procenty_DB".inJednostkaKwaśna,
	//                  inPrzewodnośćCzystejWody := "ms_na_procenty_DB".inPrzewodnośćCzystejWody,
	//                  inWartośćOdcięcia        := 0.3,
	//                  inJestMycieKwaśne        := ("CIP1_RecepturyStacjaMycia".numerKrokuMycia = 4),
	//                  inJestMycieAlkaliczne    := ("CIP1_RecepturyStacjaMycia".numerKrokuMycia = 3),
	//                  outStężenieŚrodka        => "ms_na_procenty_DB".outStężenieŚrodkaTor1);
	
	// //milisimensy na procenty Tor2
	// "ms_na_procenty"(inWartośćMierzona        := "CIP2_obiekty".obiekt["C101CT21"].WartośćPomiaru,
	//                  inJednostkaAlkaliczna    := "ms_na_procenty_DB".inJednostkaAlkaliczna,
	//                  inJednostkaKwaśna        := "ms_na_procenty_DB".inJednostkaKwaśna,
	//                  inPrzewodnośćCzystejWody := "ms_na_procenty_DB".inPrzewodnośćCzystejWody,
	//                  inWartośćOdcięcia        := 0.3,
	//                  inJestMycieKwaśne        := ("CIP2_RecepturyStacjaMycia".numerKrokuMycia = 4),
	//                  inJestMycieAlkaliczne    := ("CIP2_RecepturyStacjaMycia".numerKrokuMycia = 3),
	//                  outStężenieŚrodka        => "ms_na_procenty_DB".outStężenieŚrodkaTor2);
	
	
	// "CIP1_obiekty".obiekt[20].pid_PV := "ms_na_procenty_DB".outStężenieŚrodkaTor1;
	
	// "CIP2_obiekty".obiekt[20].pid_PV := "ms_na_procenty_DB".outStężenieŚrodkaTor2;
	
	
	
	// //lampka zielona
	// IF "CIP1_program".program.numerKroku > 7100 OR
	//     "CIP2_program".program.numerKroku > 7100 THEN
	//     "doLmpkaZielona" := 1;
	// ELSE
	//     "doLmpkaZielona" := 0;
	// END_IF;
	// IF "CIP1_hmi".button.bPauza.set THEN
	//     "doLmpkaZielona" := "Clock_2Hz";
	// END_IF;
	
	// REGION lampki
	//     //lampka czerwona
	//     IF "diKSB_1" = 0 OR "diKSB_2" = 0 OR "awaria" OR "awaria2" THEN
	//         "doLampkaCzerwona" := "Clock_5Hz";
	//     END_IF;
	    
	//     "suma" := 0;
	//     FOR "x" := 2 TO 14 DO
	//         IF "CIP1_alarmy".alarm["x"].stan > 0 THEN
	//             "suma" := "suma" + 1;
	//         END_IF;
	//     END_FOR;
	    
	    
	//     IF "suma" > 0 THEN
	//         "awaria" := 1;
	//     ELSE
	//         "awaria" := 0;
	//     END_IF;
	    
	    
	//     "suma2" := 0;
	//     FOR "x2" := 2 TO 14 DO
	//         IF "CIP2_alarmy".alarm["x2"].stan > 0 THEN
	//             "suma2" := "suma2" + 1;
	//         END_IF;
	//     END_FOR;
	    
	    
	//     IF "suma2" > 0 THEN
	//         "awaria2" := 1;
	//     ELSE
	//         "awaria2" := 0;
	//     END_IF;
	    
	// END_REGION
	// "rec_circuit_aq" := 445 * ("CIP1_RecepturyStacjaMycia".numerKrokuMycia);
	// "rec_program_aq"  := 445 * ("CIP1_RecepturyStacjaMycia".numerUżywanejReceptury);
	// IF
	//     "CIP1_program".program.numerKroku = 7200 THEN
	//     "rec_circuit" := 1;
	//     "rec_program" := 1;
	// END_IF;
	// IF
	//     "CIP1_program".program.numerKroku > 7200 THEN
	//     "rec_cipRun" := 1;
	//     "rec_circuit" := 1;
	//     "rec_program" := 1;
	// END_IF;
	
	// "rec2_circuit_aq" := 445 * ("CIP2_RecepturyStacjaMycia".numerKrokuMycia);;
	// "rec_program_aq(1)":=445*"CIP2_RecepturyStacjaMycia".numerUżywanejReceptury;
	
	// IF
	//     "CIP2_program".program.numerKroku = 7200 THEN
	//     "rec_circuit2" := 1;
	//     "rec_program2" := 1;
	// END_IF;
	// IF
	//     "CIP2_program".program.numerKroku > 7200 THEN
	//     "rec_cipRun2" := 1;
	//     "rec_circuit2" := 1;
	//     "rec_program2" := 1;
	// END_IF;
	// // "rec_program_aq" := 2000;
	
	
	
	
	
	
	
END_FUNCTION

FUNCTION "Tor0.procedury_obiektów" : Void
{ S7_Optimized_Access := 'TRUE' }
VERSION : 0.1
   VAR_TEMP 
      obj : Int;
      nr : Int;
      Mnr : String;
      aktualnyNumerReceptury : Int;
      aktualnyKrokMycia : Int;
      temp : Int;
   END_VAR


BEGIN
	    //program zawiera procedury dla napedów i zaworów dla procedur o numerze >1  (procedura 0 i 1 jest obsługiwana w programie Obsługa obiektów)
	    //procedury wyzwalane  z progrmu TablicaProcedór dla kolejnych kroków  "F1".obiekt["F100CP01"].procedura: = 2
	    //wyzwolenie procedury zero  automatycznie  wyłącza naped/zawór
	    //procedura:=1   uruchamia napęd/zawór na 100% - czyli załaczenie napedu jak kiedyś SET -- obsługiwana jest w programie Obsługa obiektów
	    //PAUZA może być obsługiwana w każdej procedurze z osobna
	    //
	    //open ctrl+shift+(*)Numeric
	    //close ctrl+shift+(/)Numeric
	
	    
	
	    
	    REGION POMPKA PODAWANIA ŁUGU W LINIE
	    
	        #nr := "Cip".tor[0].pompkaDozowaniaŁuguwLinię;
	        
	        CASE "Tor1_program".program.numerKroku OF
	            7100..7699:  //we wszystkich krokach
	                "Cip".obiekt[#nr].procedura := 2;
	            ELSE
	                "Cip".obiekt[#nr].procedura := 0;
	        END_CASE;
	        
	    CASE "Cip".obiekt[#nr].procedura OF
	    2:
	    //set - warunki dla wejścia funkcji Set
	    "Cip".obiekt[#nr].SetReset.czasDoSet := 10;
	    "Cip".obiekt[#nr].SetReset.inSet :=
	    "Cip".obiekt["Cip".tor[0].zbiorniczekDozowaniaŁugu.czujnikDolnegoPoziomu].hmiPotwWysterowania = 1
	    AND "Cip".obiekt["Cip".tor[1].zawórDozowaniaLuguwLinię].hmiPotwWysterowania=1;
	    
	    //reset - warunki dla wejścia funkcji Reset
	    "Cip".obiekt[#nr].SetReset.czasDoReset := 0;
	    "Cip".obiekt[#nr].SetReset.inReset :=
	    "Cip".obiekt["Cip".tor[0].zbiorniczekDozowaniaŁugu.czujnikDolnegoPoziomu].hmiPotwWysterowania = 0
	    OR "Cip".obiekt["Cip".tor[1].zawórDozowaniaLuguwLinię].hmiPotwWysterowania=0;
	    
	    //załaczanie
	    "Cip".obiekt[#nr].inStartAuto := "Cip".obiekt[#nr].SetReset.wyjście;
	    
	    //wysterowanie
	    "Cip".obiekt[#nr].inZadaneWysterowanieAuto := 100.0;
	    
	    
	    //wysterowanie
	    "Cip".obiekt[#nr].inZadaneWysterowanieAuto := 100.0;
	    END_CASE;
	    END_REGION
	    
	    REGION POMPKA DOZOWANIA KWASU W LINIE
	    
	        #nr := "Cip".tor[0].pompkaDozowaniaKwasuwLinię;
	        CASE "Tor1_program".program.numerKroku OF
	            7100..7699:  //we wszystkich krokach
	                "Cip".obiekt[#nr].procedura := 2;
	            ELSE
	                "Cip".obiekt[#nr].procedura := 0;
	        END_CASE;
	        
	    CASE "Cip".obiekt[#nr].procedura OF
	    2:
	    //set - warunki dla wejścia funkcji Set
	    "Cip".obiekt[#nr].SetReset.czasDoSet := 10;
	    "Cip".obiekt[#nr].SetReset.inSet :=
	    "Cip".obiekt["Cip".tor[0].zbiorniczekDozowaniaKwasu.czujnikDolnegoPoziomu].hmiPotwWysterowania = 1
	    AND
	    ("Cip".obiekt["Cip".tor[1].zawórDozowaniaKwasuwLinię].hmiPotwWysterowania = 1
	    OR "Cip".obiekt["Cip".tor[2].zawórDozowaniaKwasuwLinię].hmiPotwWysterowania = 1);
	    
	    
	    //reset - warunki dla wejścia funkcji Reset
	    "Cip".obiekt[#nr].SetReset.czasDoReset := 0;
	    "Cip".obiekt[#nr].SetReset.inReset :=
	    "Cip".obiekt["Cip".tor[0].zbiorniczekDozowaniaKwasu.czujnikDolnegoPoziomu].hmiPotwWysterowania = 0
	    OR "Cip".obiekt["Cip".tor[1].zawórDozowaniaKwasuwLinię].hmiPotwWysterowania = 0;
	    
	    //załaczanie
	    "Cip".obiekt[#nr].inStartAuto := "Cip".obiekt[#nr].SetReset.wyjście;
	    
	    //wysterowanie
	    "Cip".obiekt[#nr].inZadaneWysterowanieAuto := 100.0;
	    
	    END_CASE;
	    
	    END_REGION
	    
	    REGION ZAWOR UZUPELNIANIA WODĄ WODY CZYSTEJ
	        
	        #nr := "Cip".tor[0].zawórUzupełnianiaWodyCzystejZbWodyCzystej;
	        
	        CASE "Tor1_program".program.numerKroku OF
	            7100..7700:
	                "Cip".obiekt[#nr].procedura := 2;
	            ELSE
	                "Cip".obiekt[#nr].procedura := 0;
	                
	        END_CASE;
	        
	        
	        
	        CASE "Cip".obiekt[#nr].procedura OF
	                
	            2:
	                //wyzwolenie timerków
	                "Cip".obiekt[#nr].SetReset.czasDoSet := 1;
	                "Cip".obiekt[#nr].SetReset.inSet :=
	                NOT "Cip".obiekt["Cip".tor[0].zbiornikwodyCzystej.czujnikDolnegoPoziomu].hmiPotwWysterowania;
	                
	                
	                "Cip".obiekt[#nr].SetReset.czasDoReset := 0;
	                "Cip".obiekt[#nr].SetReset.inReset :=
	                "Cip".obiekt["Cip".tor[0].zbiornikwodyCzystej.czujnikGórnegoPoziomu].hmiPotwWysterowania;
	                
	                //załaczanie
	                "Cip".obiekt[#nr].inStartAuto := "Cip".obiekt[#nr].SetReset.wyjście;
	                
	        END_CASE;
	    END_REGION
	    
	    REGION ZAWOR UZUPELNIANIA WODĄ zbiornika ługu
	        
	        #nr := "Cip".tor[0].zawórUzupełnianiaWodyCzystejZbŁugu;
	        
	        CASE "Tor1_program".program.numerKroku OF
	            7100..7700:
	                "Cip".obiekt[#nr].procedura := 2;
	            ELSE
	                "Cip".obiekt[#nr].procedura := 0;
	                
	        END_CASE;
	        
	        
	        
	        CASE "Cip".obiekt[#nr].procedura OF
	                
	            2:
	                //wyzwolenie timerków
	                "Cip".obiekt[#nr].SetReset.czasDoSet := 1;
	                "Cip".obiekt[#nr].SetReset.inSet :=
	                NOT "Cip".obiekt["Cip".tor[0].zbiornikŁugu.czujnikDolnegoPoziomu].hmiPotwWysterowania;
	                
	                
	                "Cip".obiekt[#nr].SetReset.czasDoReset := 5;
	                "Cip".obiekt[#nr].SetReset.inReset :=
	                "Cip".obiekt["Cip".tor[0].zbiornikŁugu.czujnikDolnegoPoziomu].hmiPotwWysterowania;
	                
	                //załaczanie
	                "Cip".obiekt[#nr].inStartAuto := "Cip".obiekt[#nr].SetReset.wyjście
	                AND NOT "Cip".obiekt["Cip".tor[0].zbiornikŁugu.czujnikGórnegoPoziomu].hmiPotwWysterowania;
	                
	        END_CASE;
	    END_REGION
	    
	    REGION ZAWOR UZUPELNIANIA WODĄ zbiornika kwasu
	        
	        #nr := "Cip".tor[0].zawórUzupełnianiaWodyCzystejZbKwasu;
	        
	        CASE "Tor1_program".program.numerKroku OF
	            7100..7700:
	                "Cip".obiekt[#nr].procedura := 2;
	            ELSE
	                "Cip".obiekt[#nr].procedura := 0;
	                
	        END_CASE;
	        
	        
	        
	        CASE "Cip".obiekt[#nr].procedura OF
	                
	            2:
	                //wyzwolenie timerków
	                "Cip".obiekt[#nr].SetReset.czasDoSet := 1;
	                "Cip".obiekt[#nr].SetReset.inSet :=
	                NOT "Cip".obiekt["Cip".tor[0].zbiornikKwasu.czujnikDolnegoPoziomu].hmiPotwWysterowania;
	                
	                
	                "Cip".obiekt[#nr].SetReset.czasDoReset := 5;
	                "Cip".obiekt[#nr].SetReset.inReset :=
	                "Cip".obiekt["Cip".tor[0].zbiornikKwasu.czujnikDolnegoPoziomu].hmiPotwWysterowania;
	                
	                //załaczanie
	                "Cip".obiekt[#nr].inStartAuto := "Cip".obiekt[#nr].SetReset.wyjście
	                AND NOT "Cip".obiekt["Cip".tor[0].zbiornikKwasu.czujnikGórnegoPoziomu].hmiPotwWysterowania;
	                
	        END_CASE;
	    END_REGION
END_FUNCTION

FUNCTION "ms_na_procenty" : Void
TITLE = przeliczanie ms na procenty roztworu mycia kwasu i ługu
{ S7_Optimized_Access := 'TRUE' }
AUTHOR : 'P.Kowalski'
VERSION : 0.1
   VAR_INPUT 
      inWartośćMierzona : Real;   // Wartość mierzona roztworu (alkalicznego lub kwaśnego) w milisimensach
      inJednostkaAlkaliczna : Real;   // 1% środka alkalicznego= 48mS
      inJednostkaKwaśna : Real;   // 1% środka kwaśnego=56mS
      inPrzewodnośćCzystejWody : Real;   // Przewodność czystej wody=0.3mS
      inWartośćOdcięcia : Real;   // Jeżeli wartość mierzona spadnie ponizej odcięcia to wyswietlamy 0
      inJestMycieKwaśne : Bool;   // obliczamy wartości podczas mycia kwaśnego
      inJestMycieAlkaliczne : Bool;   // obliczamy wartości podczas mycia alkalicznego
   END_VAR

   VAR_OUTPUT 
      outStężenieŚrodka : Real;
   END_VAR

   VAR_TEMP 
      temp_1 : Real;
      temp_2 : Real;
      temp_3 : Real;
      temp_4 : Real;
      temp_5 : Real;
   END_VAR


BEGIN
	    // Nastawa:                    Wartość:
	    //  1:  1% środka alkalicznego= 48  mS
	    //  2:  1% środka kwaśnego= 56  mS
	    //  3:  Przewodność czystej wody    0,3 mS
	    // -------------------------------------------------  
	    //     Obliczenia:
	    // ---------------
	    //     Wartość mierzona roztworu alkalicznego[mS]:
	    //     72  mS
	    //     Stężenie środka alkalicznego [%]:
	    //     x=72/48     -Tu jest formuła
	    //     1,5 %   Wskazania DO wyświetlenia w kroku 3 programu stacji mycia
	    //     Wartość stężenia procentowego środka alkaliczengo wyświetlamy na panelu obok wartości mierzonej w mSiemensach - nie używamy jej nigdzie w programie, tylko wyświetlamy w kroku 3
	    // ---------------
	    //     Wartość mierzona roztworu kwaśnego[mS]:
	    //     57  mS
	    //     Stężenie środka kwaśnego [%]:
	    //      x=57/56     -Tu jest formuła
	    //     1,0 %   Wskazania DO wyświetlenia w kroku 4 programu stacji mycia
	    //    -------------
	    //     Jeżeli wartość mierzona spadnie ponizej
	    //     przewodnosc wody+ wartosc odciecia =0,6 mS
	    //     wpisujemy stężenie 0%
	    //     Wartość stężenia procentowego środka kwasnego wyświetlamy na panelu obok wartości mierzonej w mSiemensach - nie używamy jej nigdzie w programie, tylko wyświetlamy w kroku 4
	    //     W pozostałych krokach wyświetlamy 0,0%
	    //     ---------------------     
	    //     Wartość tą należy też dodać DO rejestracji w InTouch dla obu torów stacji mycia.
	    //     
	    
	IF #inJestMycieAlkaliczne THEN
	    #outStężenieŚrodka := #inWartośćMierzona / (#inJednostkaAlkaliczna+0.000001);
	END_IF;
	
	IF #inJestMycieKwaśne THEN
	    #outStężenieŚrodka := #inWartośćMierzona / (#inJednostkaKwaśna+0.000001);
	END_IF;
	
	IF #inWartośćMierzona < #inPrzewodnośćCzystejWody + 0.3 THEN
	    #outStężenieŚrodka := 0;
	END_IF;
	
	IF #inJestMycieAlkaliczne = 0 AND #inJestMycieKwaśne = 0 THEN
	    #outStężenieŚrodka := 0.0;
	END_IF;
	
	
END_FUNCTION

FUNCTION_BLOCK "FB_RecepturyStacjaMycia"
{ S7_Optimized_Access := 'TRUE' }
VERSION : 0.1
   VAR 
      numerWyswietlanejReceptury : Int := 1;   // nowy numer receptury powoduje odcvzytanie receptury  o nowym numerze i skopiowanie do receptury 0
      staryNumerWyswietlanejReceptury : Int := 1;   // stary numer do kontroli triggera wspisywania nowego numeru
      "klawiszReceptura+1" : Bool := FALSE;
      "klawiszReceptura-1" : Bool := FALSE;
      numerUżywanejReceptury : Int := 1;   // numer używanej receptury
      klawiszKopiujRecepturę : Bool := FALSE;   // kopiuje recepture 0 do receptury 99
      klawiszWklejSkopiowanąRecepturę : Bool := FALSE;   // kopiuje recepture 99 do wyswietlanej receptury
      klawiszZapiszRecepturę : Bool := FALSE;   // zapisuje receprure wyswietlaną  rec 0 do receptury o wybranym numerze
      klawiszUżyjTejReceptury : Bool := FALSE;   // klawisz wpisuje do programu numer uzytej receptury
      numerKrokuMycia : Int := 0;   // krok mycia- numer kroku receptury dodatkowo wpisywany w krokach mycia
      numerWyswietlanegoKroku : Int;
      staryNumerWyswietlanegoKroku : Int;
      "klawiszKrok+1" : Bool;
      "klawiszKrok-1" : Bool;
      "___" : Bool := FALSE;
      bPokazOknoWyboruReceptury : Bool := FALSE;   // sygnał do HMI żeby pokazać okno tabelę wyboru receptury
   END_VAR
   VAR RETAIN
      Receptura : Array[0..20] of "typRecepturaStacjiMycia";
   END_VAR
   VAR 
      "receptura-1" {InstructionName := 'R_TRIG'; LibVersion := '1.0'} : R_TRIG;
      "receptura+1" {InstructionName := 'R_TRIG'; LibVersion := '1.0'} : R_TRIG;
      wybór_recept {InstructionName := 'R_TRIG'; LibVersion := '1.0'} : R_TRIG;
      kopiuj {InstructionName := 'R_TRIG'; LibVersion := '1.0'} : R_TRIG;
      wklej {InstructionName := 'R_TRIG'; LibVersion := '1.0'} : R_TRIG;
      zapisz {InstructionName := 'R_TRIG'; LibVersion := '1.0'} : R_TRIG;
      użyj {InstructionName := 'R_TRIG'; LibVersion := '1.0'} : R_TRIG;
      "krok+" {InstructionName := 'R_TRIG'; LibVersion := '1.0'} : R_TRIG;
      "krok-" {InstructionName := 'R_TRIG'; LibVersion := '1.0'} : R_TRIG;
      wybór_kroku {InstructionName := 'R_TRIG'; LibVersion := '1.0'} : R_TRIG;
      licznik_1 { S7_SetPoint := 'True'} : Int;   // taki liczniczek w razie co
      licznikDoAlarmu : Real;
   END_VAR


BEGIN
	//program służy do zasilenia receptury [0] która jest wyswietlana
	//i do kopiowania i zapisu receptur /kopia do receptury 20
	
	
	
	REGION //obsługa klawiszy receptura +  receptura-
	    #"receptura-1"(CLK := #"klawiszReceptura-1");
	    #"receptura+1"(CLK := #"klawiszReceptura+1");
	    IF #numerWyswietlanejReceptury < 1 THEN
	        #numerWyswietlanejReceptury := #staryNumerWyswietlanejReceptury;
	    END_IF;
	    IF #numerWyswietlanejReceptury > 19 THEN
	        #numerWyswietlanejReceptury := #staryNumerWyswietlanejReceptury;
	    END_IF;
	    IF #"receptura-1".Q = 1 AND #numerWyswietlanejReceptury > 1 THEN
	        #numerWyswietlanejReceptury := #numerWyswietlanejReceptury - 1;
	        ;
	    END_IF;
	    IF #"receptura+1".Q = 1 AND #numerWyswietlanejReceptury < 19 THEN
	        #numerWyswietlanejReceptury := #numerWyswietlanejReceptury + 1;
	        ;
	    END_IF;
	END_REGION
	
	
	REGION //obsługa klawiszy krok +  krok-
	    #"krok-"(CLK := #"klawiszKrok-1");
	    #"krok+"(CLK := #"klawiszKrok+1");
	    IF #numerWyswietlanegoKroku < 1 THEN
	        #numerWyswietlanegoKroku := 1;
	    END_IF;
	    IF #numerWyswietlanegoKroku > 6 THEN
	        #numerWyswietlanegoKroku := 6;
	    END_IF;
	    IF #"krok-".Q = 1 AND #numerWyswietlanegoKroku > 1 THEN
	        #numerWyswietlanegoKroku := #numerWyswietlanegoKroku - 1;
	        ;
	    END_IF;
	    IF #"krok+".Q = 1 AND #numerWyswietlanegoKroku < 6 THEN
	        #numerWyswietlanegoKroku := #numerWyswietlanegoKroku + 1;
	        ;
	    END_IF;
	END_REGION
	
	REGION //gdy ktoś zmieni numer receptury to przepisz zawartość wybranej do receptury 0 (wyświetlanej na panelu)
	    #wybór_recept(CLK := (#numerWyswietlanejReceptury <> #staryNumerWyswietlanejReceptury));
	    IF #wybór_recept.Q THEN
	        #Receptura[0] := #Receptura[#numerWyswietlanejReceptury];
	        #Receptura[0].nazwaReceptury:=#Receptura[#numerWyswietlanejReceptury].nazwaReceptury;
	        
	        
	    END_IF;
	    #staryNumerWyswietlanejReceptury := #numerWyswietlanejReceptury;
	    
	    IF #wybór_recept.Q THEN
	        #numerWyswietlanegoKroku:= 1;
	        #staryNumerWyswietlanegoKroku := 1;
	        #Receptura[0].Krok[0] := #Receptura[0].Krok[#numerWyswietlanegoKroku];
	    END_IF;
	END_REGION
	
	
	
	
	REGION //gdy ktoś zmieni numer kroku to przepisz zawartość wybranego kroku do kroku 0 (wyświetlanego na panelu)
	    #wybór_kroku(CLK := (#numerWyswietlanegoKroku <> #staryNumerWyswietlanegoKroku));
	    
	    // IF #wybór_kroku.Q THEN
	    //     #Receptura[0].Krok[#staryNumerWyswietlanegoKroku] := #Receptura[0].Krok[0];
	    // END_IF;
	    
	    IF #wybór_kroku.Q THEN
	        #Receptura[0].Krok[0] := #Receptura[0].Krok[#numerWyswietlanegoKroku];
	    END_IF;
	    
	    #staryNumerWyswietlanegoKroku := #numerWyswietlanegoKroku;
	END_REGION
	
	
	
	REGION //operacje kopiuj wklej uzyj
	    #kopiuj(CLK := #klawiszKopiujRecepturę);
	    IF #kopiuj.Q THEN
	        #Receptura[20] := #Receptura[0];
	    END_IF;
	    
	    #wklej(CLK := #klawiszWklejSkopiowanąRecepturę);
	    IF #wklej.Q THEN
	        #Receptura[0] := #Receptura[20];
	        // "RecepturyMycia".Receptura[0] := "RecepturyMycia".Receptura["RecepturyMycia".numerWyswietlanejReceptury];
	    END_IF;
	    
	    #zapisz(CLK := #klawiszZapiszRecepturę);
	    
	    IF #zapisz.Q THEN // AND #krokMycia = 0   --zapis mozliwy tylko gdy nie wykonuje sie mycie
	        #Receptura[0].Krok[#numerWyswietlanegoKroku] := #Receptura[0].Krok[0];
	        
	        #Receptura[#numerWyswietlanejReceptury] := #Receptura[0];
	        
	    END_IF;
	    
	    #użyj(CLK := #klawiszUżyjTejReceptury);
	    IF #użyj.Q THEN
	        #numerUżywanejReceptury := #numerWyswietlanejReceptury;
	    END_IF;
	END_REGION
	
	//kasowanie tymczasowych
	//
	#"klawiszReceptura-1" := 0;
	#"klawiszReceptura+1" := 0;
	#klawiszKopiujRecepturę := 0;
	#klawiszWklejSkopiowanąRecepturę := 0;
	#klawiszZapiszRecepturę := 0;
	#"klawiszKrok+1" := 0;
	#"klawiszKrok-1" := 0;
	//opuznienie kasowania klawisza wybrania receptury ,zeby program nadrzedny
	//zdazyl zauwazyc stan tego klawisza w HMi klawisz ma być typu set
	IF #klawiszUżyjTejReceptury = 1 THEN
	    
	    #licznik_1:=
	    #licznik_1+1;
	    
	    IF #licznik_1 > 5 THEN
	        #klawiszUżyjTejReceptury := 0;
	        #licznik_1 := 0;
	    END_IF;
	    
	END_IF;
	
	
	
END_FUNCTION_BLOCK

FUNCTION_BLOCK "Flipaj_FB"
{ S7_Optimized_Access := 'TRUE' }
VERSION : 0.1
   VAR_INPUT 
      in { ExternalAccessible := 'False'; ExternalVisible := 'False'; ExternalWritable := 'False'} : Bool;
      ile_petli { ExternalAccessible := 'False'; ExternalVisible := 'False'; ExternalWritable := 'False'} : Int;   // że filpanie ma dziać się w kółko
      start_od_zera { ExternalAccessible := 'False'; ExternalVisible := 'False'; ExternalWritable := 'False'} : Bool;   // że po wyzwoleniu jest najpierw OFF
      czas_ON { ExternalAccessible := 'False'; ExternalVisible := 'False'; ExternalWritable := 'False'} : Int;   // czas załączenia wyjścia 0.1 s
      czas_OFF { ExternalAccessible := 'False'; ExternalVisible := 'False'; ExternalWritable := 'False'} : Int;   // czas wyłączenia wyjścia 0.1s
   END_VAR

   VAR_OUTPUT 
      Q { ExternalAccessible := 'False'; ExternalVisible := 'False'; ExternalWritable := 'False'} : Bool;
   END_VAR

   VAR 
      licznik { ExternalAccessible := 'False'; ExternalVisible := 'False'; ExternalWritable := 'False'} : LInt;
      licznik_petli { ExternalAccessible := 'False'; ExternalVisible := 'False'; ExternalWritable := 'False'} : Int;
   END_VAR


BEGIN
	        IF #licznik > (#licznik_petli+1) * (#czas_ON + #czas_OFF) THEN
	            #in := 0;
	        END_IF;
	
	IF #in THEN
	    #licznik := #licznik + 1;
	ELSE
	    #licznik := 0;
	    #Q:=0;
	    #licznik_petli := 0;
	END_IF;
	
	
	    
	IF #start_od_zera=1 THEN
	    IF #licznik > 0 + ((#czas_ON + #czas_OFF) * #licznik_petli)
	        AND #licznik <= #czas_OFF + ((#czas_ON + #czas_OFF) * #licznik_petli) THEN
	        #Q := 0;
	    END_IF;
	    
	    IF (#licznik > #czas_OFF + ((#czas_ON + #czas_OFF) * #licznik_petli))
	        AND #licznik <= (#czas_ON + #czas_OFF + ((#czas_ON + #czas_OFF) * #licznik_petli)) THEN
	        #Q := 1;
	    END_IF;
	    
	    IF #licznik = (#czas_ON + #czas_OFF + ((#czas_ON + #czas_OFF) * #licznik_petli)) THEN
	        #licznik_petli := #licznik_petli + 1;
	    END_IF;
	END_IF;
	        
	IF #start_od_zera=0 THEN
	    IF #licznik > 0 + ((#czas_ON + #czas_OFF) * #licznik_petli)
	        AND #licznik <= #czas_ON + ((#czas_ON + #czas_OFF) * #licznik_petli) THEN
	        #Q := 1;
	    END_IF;
	    
	    IF (#licznik > #czas_ON+ ((#czas_ON + #czas_OFF) * #licznik_petli))
	        AND #licznik <= (#czas_ON + #czas_OFF + ((#czas_ON + #czas_OFF) * #licznik_petli)) THEN
	        #Q := 0;
	    END_IF;
	    
	    IF #licznik = (#czas_ON + #czas_OFF + ((#czas_ON + #czas_OFF) * #licznik_petli)) THEN
	        #licznik_petli := #licznik_petli + 1;
	    END_IF;
	END_IF;
	        
	        IF #licznik_petli >= #ile_petli THEN
	            #Q := 0;
	    
	        END_IF;
	    
	  
	
END_FUNCTION_BLOCK

FUNCTION_BLOCK "FB_obsluga_alarmow"
{ S7_Optimized_Access := 'TRUE' }
VERSION : 0.1
   VAR_INPUT 
      aktualnyIndexProgramu { ExternalAccessible := 'False'; ExternalVisible := 'False'; ExternalWritable := 'False'} : Int;
   END_VAR

   VAR 
      alarm { S7_SetPoint := 'False'} : Array[0..99] of "typAlarmNew";   // instancje nazwij np. F1.alarmy
      x { ExternalAccessible := 'False'; ExternalVisible := 'False'; ExternalWritable := 'False'} : Int;
   END_VAR


BEGIN
	//program obsługuje obiekty rozpoznaje ich typy i wykonuje odpowiednie akcje
	//zeruje timery
	//przelicza wartości
	//wykonuje procedure [0] i [1] dla każdego obiektu
	
	
	FOR #x := 1 TO 99 DO
	
	    
	    // IF #alarm[#x].procedura = 0 THEN //jezeli aktualna procedura 0 to kasuj alarm
	    //     #alarm[#x].timerek := 0;
	    //     #alarm[#x].stan := 0;
	    // END_IF;
	    
	    IF #alarm[#x].procedura = 1 THEN //jezeli aktualna procedura 1 to wlacz alarm
	        #alarm[#x].timerek := 0;
	        #alarm[#x].stan := 1;
	    END_IF;
	END_FOR;
	
	
	
	
	
	
	
	
	
	
	
	
	
END_FUNCTION_BLOCK

FUNCTION_BLOCK "FB_obsluga_obiektow"
{ S7_Optimized_Access := 'TRUE' }
VERSION : 0.1
   VAR 
      obiekt { S7_SetPoint := 'False'} : Array[0..110] of "typObiekt";   // instancje nazwij np.C1 dla stacji CIP1
      tor { S7_SetPoint := 'False'} : Array[0..2] of "typFunkcjeObiektówCipu";   // [0..xx] ilosc torów stacji CIP, 0- tor wspólny
      x { ExternalAccessible := 'False'; ExternalVisible := 'False'; ExternalWritable := 'False'} : Int;
   END_VAR


BEGIN
	//program obsługuje obiekty rozpoznaje ich typy i wykonuje odpowiednie akcje
	//zeruje timery
	//przelicza wartości
	//wykonuje procedure [0] i [1] dla każdego obiektu
	
	
	
	FOR #x := 1 TO 110 DO
	    CASE #obiekt[#x].typObiektu OF
	            
	            
	        1:    //zawór przełączny "Banjo" "MixProof" i inne ON OFF    
	            REGION typ1
	                
	                
	                IF #obiekt[#x].hmiTrybAutoManual THEN
	                    #obiekt[#x].outStartUrządzenie := #obiekt[#x].hmiManualStart AND #obiekt[#x].inZezwolenieNaPracę; //jeżeli tryb ręczny to steruj zawór ze stacyjki
	                ELSE
	                    #obiekt[#x].outStartUrządzenie := #obiekt[#x].inStartAuto AND #obiekt[#x].inZezwolenieNaPracę;
	                END_IF;
	                
	                //obsługa potwierdzeń otwarcia zamknięcia zaworu
	                IF #obiekt[#x].inJestPotwWysterowania THEN
	                    #obiekt[#x].hmiPotwWysterowania := #obiekt[#x].diPotwWysterowania;
	                ELSE
	                    #obiekt[#x].hmiPotwWysterowania := #obiekt[#x].outStartUrządzenie;
	                END_IF;
	                IF #obiekt[#x].inJestPotwNiewysterowania THEN
	                    #obiekt[#x].hmiPotwNieWysterowania := #obiekt[#x].diPotwNieWysterowania;
	                ELSE
	                    #obiekt[#x].hmiPotwNieWysterowania := NOT #obiekt[#x].outStartUrządzenie;
	                END_IF;
	                
	                
	                
	                //SYMULACJA
	                //
	                IF #obiekt[#x].hmiSymulujSygnałyWejsciowe THEN
	                    #obiekt[#x].hmiPotwWysterowania := #obiekt[#x].outStartUrządzenie;
	                    #obiekt[#x].hmiPotwNieWysterowania := NOT #obiekt[#x].outStartUrządzenie;
	                END_IF;
	                
	                //obsługa LiftUp Lift Down w zaworze Mixproof
	                //
	                IF #obiekt[#x].hmiTrybAutoManual THEN
	                    #obiekt[#x].outLiftUp := #obiekt[#x].hmiManualLiftUp AND #obiekt[#x].inZezwolenieNaPracę; //jeżeli tryb ręczny to steruj zawór ze stacyjki
	                ELSE
	                    #obiekt[#x].outLiftUp := #obiekt[#x].inLiftUp AND #obiekt[#x].inZezwolenieNaPracę;
	                END_IF;
	                IF #obiekt[#x].hmiTrybAutoManual THEN
	                    #obiekt[#x].outLiftDown := #obiekt[#x].hmiManualLiftDown AND #obiekt[#x].inZezwolenieNaPracę; //jeżeli tryb ręczny to steruj zawór ze stacyjki
	                ELSE
	                    #obiekt[#x].outLiftDown := #obiekt[#x].inLiftDown AND #obiekt[#x].inZezwolenieNaPracę;
	                END_IF;
	                
	                
	                
	                // zliczanie czasu awarii gdy nie ma potwierdzenia 
	                IF #obiekt[#x].outStartUrządzenie AND NOT #obiekt[#x].hmiPotwWysterowania
	                    AND #obiekt[#x].czasDoAwariiPV < 10000 THEN
	                    #obiekt[#x].czasDoAwariiPV := #obiekt[#x].czasDoAwariiPV + 1;
	                END_IF;
	                IF NOT #obiekt[#x].outStartUrządzenie AND NOT #obiekt[#x].hmiPotwNieWysterowania
	                    AND #obiekt[#x].czasDoAwariiPV < 10000 THEN
	                    #obiekt[#x].czasDoAwariiPV := #obiekt[#x].czasDoAwariiPV + 1;
	                END_IF;
	                // wystawienie sygnału awarii
	                IF #obiekt[#x].czasDoAwariiPV > #obiekt[#x].czasDoAwariiSP THEN
	                    #obiekt[#x].Awaria := 1;
	                ELSE
	                    #obiekt[#x].Awaria := 0;
	                END_IF;
	                // kasowanie czasu awarii gdy wszystkie potwierdzenia są ok
	                IF #obiekt[#x].outStartUrządzenie AND #obiekt[#x].hmiPotwWysterowania
	                THEN
	                    #obiekt[#x].czasDoAwariiPV := 0;
	                END_IF;
	                IF NOT #obiekt[#x].outStartUrządzenie AND #obiekt[#x].hmiPotwNieWysterowania
	                THEN
	                    #obiekt[#x].czasDoAwariiPV := 0;
	                END_IF;
	                IF #obiekt[#x].hmiResetAwaria
	                THEN
	                    #obiekt[#x].czasDoAwariiPV := 0;
	                    #obiekt[#x].hmiResetAwaria := 0;
	                END_IF;
	                
	                //stan zaworu grafika
	                IF #obiekt[#x].hmiTrybAutoManual = 0 THEN
	                    IF #obiekt[#x].outStartUrządzenie = 0 THEN
	                        #obiekt[#x].hmiStanUrządzenia := 1;
	                    END_IF;
	                    IF #obiekt[#x].outStartUrządzenie = 1 THEN
	                        #obiekt[#x].hmiStanUrządzenia := 3;
	                    END_IF;
	                    IF #obiekt[#x].Awaria = 1 THEN
	                        #obiekt[#x].hmiStanUrządzenia := 5;
	                    END_IF;
	                END_IF;
	                
	                
	                IF #obiekt[#x].hmiTrybAutoManual = 1 THEN
	                    IF #obiekt[#x].outStartUrządzenie = 0 THEN
	                        #obiekt[#x].hmiStanUrządzenia := 2;
	                    END_IF;
	                    IF #obiekt[#x].outStartUrządzenie = 1 THEN
	                        #obiekt[#x].hmiStanUrządzenia := 4;
	                    END_IF;
	                    IF #obiekt[#x].Awaria = 1 THEN
	                        #obiekt[#x].hmiStanUrządzenia := 6;
	                    END_IF;
	                END_IF;
	                
	                
	            END_REGION
	        2: //zawór analogowy
	            REGION typ2
	                
	                
	                
	                
	                IF #obiekt[#x].hmiTrybAutoManual THEN
	                    
	                    #obiekt[#x].outWysterowanieUrządzenia := LIMIT(MN := 0.0, IN := #obiekt[#x].hmiManualneWysterowanie, MX := 100.0); //jezeli tryb ręczny to zadane otwarcie ze stacyjki
	                    
	                    IF #obiekt[#x].hmiManualStart = 0 THEN
	                        #obiekt[#x].outWysterowanieUrządzenia := 0;
	                    END_IF;
	                    
	                    
	                ELSE
	                    #obiekt[#x].outWysterowanieUrządzenia := LIMIT(MN := 0.0, IN := #obiekt[#x].inZadaneWysterowanieAuto, MX := 100.0);
	                END_IF;
	                IF #obiekt[#x].inZezwolenieNaPracę = false THEN  //ZERUJ WYJSCIE JAK BRAK ZEZWOLENIA NA PRACĘ NA PRZYKŁAD STOP AWARJNY
	                    #obiekt[#x].outWysterowanieUrządzenia := 0.0;
	                END_IF;
	                
	                IF #obiekt[#x].outWysterowanieUrządzenia = 0 THEN
	                    #obiekt[#x].outStartUrządzenie := FALSE;
	                END_IF;
	                IF #obiekt[#x].outWysterowanieUrządzenia = 100.0 THEN
	                    #obiekt[#x].outStartUrządzenie := TRUE;
	                END_IF;
	                //obsługa potwierdzeń otwarcia zamknięcia zaworu
	                IF NOT #obiekt[#x].inJestPotwWysterowania THEN
	                    #obiekt[#x].diPotwWysterowania := #obiekt[#x].outStartUrządzenie;
	                END_IF;
	                IF NOT #obiekt[#x].inJestPotwNiewysterowania THEN
	                    #obiekt[#x].diPotwNieWysterowania := NOT #obiekt[#x].outStartUrządzenie;
	                END_IF;
	                IF #obiekt[#x].hmiSymulujSygnałyWejsciowe THEN
	                    IF #obiekt[#x].inJestPotwWysterowania THEN
	                        #obiekt[#x].diPotwWysterowania := #obiekt[#x].hmiSymulacjaPotwNieWysterowania;
	                    END_IF;
	                    IF #obiekt[#x].inJestPotwNiewysterowania THEN
	                        #obiekt[#x].diPotwNieWysterowania := #obiekt[#x].hmiSymulacjaPotwNieWysterowania;
	                    END_IF;
	                END_IF;
	                
	                // zliczanie czasu awarii gdy nie ma potwierdzenia 
	                IF #obiekt[#x].outStartUrządzenie AND NOT #obiekt[#x].diPotwWysterowania
	                    AND #obiekt[#x].czasDoAwariiPV < 10000 THEN
	                    #obiekt[#x].czasDoAwariiPV := #obiekt[#x].czasDoAwariiPV + 1;
	                END_IF;
	                IF NOT #obiekt[#x].outStartUrządzenie AND NOT #obiekt[#x].diPotwNieWysterowania
	                    AND #obiekt[#x].czasDoAwariiPV < 10000 THEN
	                    #obiekt[#x].czasDoAwariiPV := #obiekt[#x].czasDoAwariiPV + 1;
	                END_IF;
	                // wystawienie sygnału awarii
	                IF #obiekt[#x].czasDoAwariiPV > #obiekt[#x].czasDoAwariiSP THEN
	                    #obiekt[#x].Awaria := 1;
	                ELSE
	                    #obiekt[#x].Awaria := 0;
	                END_IF;
	                // kasowanie czasu awarii gdy wszystkie potwierdzenia są ok
	                IF #obiekt[#x].outStartUrządzenie AND #obiekt[#x].diPotwWysterowania
	                THEN
	                    #obiekt[#x].czasDoAwariiPV := 0;
	                END_IF;
	                IF NOT #obiekt[#x].outStartUrządzenie AND #obiekt[#x].diPotwNieWysterowania
	                THEN
	                    #obiekt[#x].czasDoAwariiPV := 0;
	                END_IF;
	                
	                
	                //grafika
	                //
	                IF #obiekt[#x].hmiTrybAutoManual =0 THEN
	                    IF (#obiekt[#x].outWysterowanieUrządzenia = 0.0) THEN
	                        #obiekt[#x].hmiStanUrządzenia := 1;
	                    END_IF;
	                    IF (#obiekt[#x].outWysterowanieUrządzenia > 0.0) THEN
	                        #obiekt[#x].hmiStanUrządzenia := 3;
	                    END_IF;
	                    IF #obiekt[#x].Awaria THEN
	                        #obiekt[#x].hmiStanUrządzenia := 6;
	                    END_IF;
	                END_IF;
	                
	                IF #obiekt[#x].hmiTrybAutoManual = 1 THEN
	                    IF (#obiekt[#x].outWysterowanieUrządzenia = 0.0) THEN
	                        #obiekt[#x].hmiStanUrządzenia := 2;
	                    END_IF;
	                    IF (#obiekt[#x].outWysterowanieUrządzenia > 0.0) THEN
	                        #obiekt[#x].hmiStanUrządzenia := 4;
	                    END_IF;
	                    IF #obiekt[#x].Awaria THEN
	                        #obiekt[#x].hmiStanUrządzenia := 6;
	                    END_IF;
	                END_IF;
	                
	                
	                
	                
	                
	                
	            END_REGION
	        3://pompa na styczniku
	            REGION typ3
	                
	                
	                
	                IF #obiekt[#x].hmiTrybAutoManual = 1 THEN
	                    #obiekt[#x].outStartUrządzenie := #obiekt[#x].hmiManualStart AND #obiekt[#x].inZezwolenieNaPracę;
	                ELSE
	                    #obiekt[#x].outStartUrządzenie := #obiekt[#x].inStartAuto AND #obiekt[#x].inZezwolenieNaPracę;
	                END_IF;
	                
	                //obsługa potwierdzeń zalaczenia
	                IF #obiekt[#x].inJestPotwWysterowania THEN
	                    #obiekt[#x].hmiPotwWysterowania := #obiekt[#x].diPotwWysterowania;
	                ELSE
	                    #obiekt[#x].hmiPotwWysterowania := #obiekt[#x].outStartUrządzenie;
	                END_IF;
	                IF #obiekt[#x].inJestPotwNiewysterowania THEN
	                    #obiekt[#x].hmiPotwNieWysterowania := #obiekt[#x].diPotwNieWysterowania;
	                ELSE
	                    #obiekt[#x].hmiPotwNieWysterowania := NOT #obiekt[#x].outStartUrządzenie;
	                END_IF;
	                
	                
	                
	                
	                
	                
	                IF #obiekt[#x].hmiSymulujSygnałyWejsciowe THEN
	                    IF #obiekt[#x].inJestPotwWysterowania THEN
	                        #obiekt[#x].hmiSymulacjaPotwWysterowania := #obiekt[#x].outStartUrządzenie;
	                    END_IF;
	                    IF #obiekt[#x].inJestPotwNiewysterowania THEN
	                        #obiekt[#x].diPotwNieWysterowania := NOT #obiekt[#x].outStartUrządzenie;
	                        ;
	                    END_IF;
	                END_IF;
	                
	                // zliczanie czasu awarii gdy nie ma potwierdzenia 
	                IF #obiekt[#x].outStartUrządzenie AND NOT #obiekt[#x].hmiPotwWysterowania
	                    AND #obiekt[#x].czasDoAwariiPV < 10000 THEN
	                    #obiekt[#x].czasDoAwariiPV := #obiekt[#x].czasDoAwariiPV + 1;
	                END_IF;
	                IF NOT #obiekt[#x].outStartUrządzenie AND NOT #obiekt[#x].hmiPotwNieWysterowania
	                    AND #obiekt[#x].czasDoAwariiPV < 10000 THEN
	                    #obiekt[#x].czasDoAwariiPV := #obiekt[#x].czasDoAwariiPV + 1;
	                END_IF;
	                // wystawienie sygnału awarii
	                IF #obiekt[#x].czasDoAwariiPV > #obiekt[#x].czasDoAwariiSP THEN
	                    #obiekt[#x].Awaria := 1;
	                ELSE
	                    #obiekt[#x].Awaria := 0;
	                END_IF;
	                // kasowanie czasu awarii gdy wszystkie potwierdzenia są ok
	                IF #obiekt[#x].outStartUrządzenie AND #obiekt[#x].hmiPotwWysterowania
	                THEN
	                    #obiekt[#x].czasDoAwariiPV := 0;
	                END_IF;
	                IF NOT #obiekt[#x].outStartUrządzenie AND #obiekt[#x].hmiPotwNieWysterowania
	                THEN
	                    #obiekt[#x].czasDoAwariiPV := 0;
	                END_IF;
	                IF #obiekt[#x].hmiResetAwaria
	                THEN
	                    #obiekt[#x].czasDoAwariiPV := 0;
	                    #obiekt[#x].hmiResetAwaria := 0;
	                END_IF;
	                
	                
	                
	                
	                
	                //zliczanie czasu pracy
	                IF #obiekt[#x].outStartUrządzenie AND #obiekt[#x].diPotwWysterowania THEN
	                    #obiekt[#x].czasPracyGodziny := #obiekt[#x].czasPracyGodziny + (1 / 36000);// dzielnik 36000 - zwiazany z cyklem wywoływania funkkcji FC Obsługa obiektów
	                END_IF;
	                
	                //grafika
	                //
	                IF #obiekt[#x].hmiTrybAutoManual = 0 THEN
	                    IF #obiekt[#x].outStartUrządzenie = 0 THEN
	                        #obiekt[#x].hmiStanUrządzenia := 1;
	                    END_IF;
	                    IF #obiekt[#x].outStartUrządzenie = 1 THEN
	                        #obiekt[#x].hmiStanUrządzenia := 3;
	                    END_IF;
	                    IF #obiekt[#x].Awaria = 1 THEN
	                        #obiekt[#x].hmiStanUrządzenia := 5;
	                    END_IF;
	                END_IF;
	                
	                
	                IF #obiekt[#x].hmiTrybAutoManual = 1 THEN
	                    IF #obiekt[#x].outStartUrządzenie = 0 THEN
	                        #obiekt[#x].hmiStanUrządzenia := 2;
	                    END_IF;
	                    IF #obiekt[#x].outStartUrządzenie = 1 THEN
	                        #obiekt[#x].hmiStanUrządzenia := 4;
	                    END_IF;
	                    IF #obiekt[#x].Awaria = 1 THEN
	                        #obiekt[#x].hmiStanUrządzenia := 6;
	                    END_IF;
	                END_IF;
	            END_REGION
	        4://Pompa na falowniku   
	            REGION typ4
	                
	                IF #obiekt[#x].hmiManualneWysterowanie > 100.0 THEN //zapobieganie przekroczeniu wpisu
	                    #obiekt[#x].hmiManualneWysterowanie := 100.0;
	                END_IF;
	                IF #obiekt[#x].hmiManualneWysterowanie < 0.0 THEN //zapobieganie przekroczeniu wpisu
	                    #obiekt[#x].hmiManualneWysterowanie := 0.0;
	                END_IF;
	                
	                IF #obiekt[#x].hmiTrybAutoManual = 1 THEN
	                    IF #obiekt[#x].outWysterowanieUrządzenia < #obiekt[#x].hmiManualneWysterowanie THEN
	                        #obiekt[#x].outWysterowanieUrządzenia := #obiekt[#x].outWysterowanieUrządzenia + (100.0 / (100 * (#obiekt[#x].pid_Rampa + 0.0001)));//rampa startu w sekundach
	                    ELSE
	                        #obiekt[#x].outWysterowanieUrządzenia := #obiekt[#x].hmiManualneWysterowanie;
	                    END_IF;
	                    #obiekt[#x].outWysterowanieUrządzenia := LIMIT(MN := 0.0, IN := #obiekt[#x].outWysterowanieUrządzenia, MX := 100.0); //jezeli tryb ręczny to zadane otwarcie ze stacyjki
	                    #obiekt[#x].outStartUrządzenie := #obiekt[#x].hmiManualStart;// AND (#obiekt[#x].outWysterowanieUrządzenia > 1.0); //AND #obiekt[#x].inZezwolenieNaPracę;
	                ELSE
	                    
	                    IF #obiekt[#x].outWysterowanieUrządzenia < #obiekt[#x].inZadaneWysterowanieAuto-5.0 THEN
	                        #obiekt[#x].outWysterowanieUrządzenia := #obiekt[#x].outWysterowanieUrządzenia + (100.0 / (100 * (#obiekt[#x].tFiltr + 0.01)));//rampa startu
	                    ELSE
	                        #obiekt[#x].outWysterowanieUrządzenia := #obiekt[#x].inZadaneWysterowanieAuto;
	                    END_IF;
	                    IF #obiekt[#x].outWysterowanieUrządzenia > #obiekt[#x].inZadaneWysterowanieAuto + 5.0 THEN
	                        #obiekt[#x].outWysterowanieUrządzenia := #obiekt[#x].outWysterowanieUrządzenia -(100.0 / (100 * (#obiekt[#x].tFiltr + 0.01)));//rampa startu
	                    ELSE
	                        #obiekt[#x].outWysterowanieUrządzenia := #obiekt[#x].inZadaneWysterowanieAuto;
	                    END_IF;
	                    
	                    #obiekt[#x].outWysterowanieUrządzenia := LIMIT(MN := 0.0, IN := #obiekt[#x].outWysterowanieUrządzenia, MX := 100.0);
	                    #obiekt[#x].outStartUrządzenie := #obiekt[#x].inStartAuto AND #obiekt[#x].inZezwolenieNaPracę;
	                END_IF;
	                
	                IF #obiekt[#x].inStartAuto = 0 AND (#obiekt[#x].hmiManualStart = 0 AND #obiekt[#x].hmiTrybAutoManual = 1) THEN//zeruj wysterowanie gdy stop
	                    #obiekt[#x].outWysterowanieUrządzenia := 0.0;
	                END_IF;
	                
	                
	                
	                //  #obiekt[#x].tagerror := UNSCALE(IN := #obiekt[#x].hmiWysterowanieFalownika, HI_LIM := 100.0, LO_LIM := 0.0, BIPOLAR := 0, OUT => #obiekt[#x].aoWysterFalownika);
	                //obsługa potwierdzeń otwarcia zamknięcia zaworu
	                IF #obiekt[#x].inJestPotwWysterowania THEN
	                    #obiekt[#x].hmiPotwWysterowania := #obiekt[#x].diPotwWysterowania;
	                ELSE
	                    #obiekt[#x].hmiPotwWysterowania := #obiekt[#x].outStartUrządzenie;
	                END_IF;
	                IF #obiekt[#x].inJestPotwNiewysterowania THEN
	                    #obiekt[#x].hmiPotwNieWysterowania := #obiekt[#x].diPotwNieWysterowania;
	                ELSE
	                    #obiekt[#x].hmiPotwNieWysterowania := NOT #obiekt[#x].outStartUrządzenie;
	                END_IF;
	                
	                
	                
	                //SYMULACJA
	                //
	                IF #obiekt[#x].hmiSymulujSygnałyWejsciowe THEN
	                    #obiekt[#x].hmiPotwWysterowania := #obiekt[#x].outStartUrządzenie;
	                    #obiekt[#x].hmiPotwNieWysterowania := NOT #obiekt[#x].outStartUrządzenie;
	                END_IF;
	                
	                // zliczanie czasu awarii gdy nie ma potwierdzenia 
	                IF #obiekt[#x].outStartUrządzenie AND NOT #obiekt[#x].hmiPotwWysterowania
	                    AND #obiekt[#x].czasDoAwariiPV < 10000 THEN
	                    #obiekt[#x].czasDoAwariiPV := #obiekt[#x].czasDoAwariiPV + 1;
	                END_IF;
	                IF NOT #obiekt[#x].outStartUrządzenie AND NOT #obiekt[#x].hmiPotwNieWysterowania
	                    AND #obiekt[#x].czasDoAwariiPV < 10000 THEN
	                    #obiekt[#x].czasDoAwariiPV := #obiekt[#x].czasDoAwariiPV + 1;
	                END_IF;
	                //wystawienie sygnału awarii
	                IF #obiekt[#x].czasDoAwariiPV > #obiekt[#x].czasDoAwariiSP THEN
	                    #obiekt[#x].Awaria := 1;
	                    
	                    ;
	                END_IF;
	                //kasowanie sygnału awarii z hmi
	                IF #obiekt[#x].hmiResetAwaria = 1 THEN
	                    #obiekt[#x].Awaria := 0;
	                    #obiekt[#x].czasDoAwariiPV := 0;
	                END_IF;
	                //kasowanie czasu awarii gdy wszystkie potwierdzenia są ok
	                IF #obiekt[#x].outStartUrządzenie AND #obiekt[#x].hmiPotwWysterowania
	                THEN
	                    #obiekt[#x].czasDoAwariiPV := 0;
	                    #obiekt[#x].Awaria := 0;
	                END_IF;
	                IF NOT #obiekt[#x].outStartUrządzenie AND #obiekt[#x].hmiPotwNieWysterowania
	                THEN
	                    #obiekt[#x].czasDoAwariiPV := 0;
	                    #obiekt[#x].Awaria := 0;
	                END_IF;
	                
	                //zliczanie czasu pracy
	                IF #obiekt[#x].outStartUrządzenie AND #obiekt[#x].diPotwWysterowania THEN
	                    #obiekt[#x].czasPracyGodziny := #obiekt[#x].czasPracyGodziny + (1 / 36000);// dzielnik 36000 - zwiazany z cyklem wywoływania funkkcji FC Obsługa obiektów
	                END_IF;
	                
	                //grafika
	                //
	                IF #obiekt[#x].hmiTrybAutoManual = 0 THEN
	                    IF #obiekt[#x].outStartUrządzenie = 0 THEN
	                        #obiekt[#x].hmiStanUrządzenia := 1;
	                    END_IF;
	                    IF #obiekt[#x].outStartUrządzenie = 1 THEN
	                        #obiekt[#x].hmiStanUrządzenia := 3;
	                    END_IF;
	                    IF #obiekt[#x].Awaria = 1 THEN
	                        #obiekt[#x].hmiStanUrządzenia := 5;
	                    END_IF;
	                END_IF;
	                
	                
	                IF #obiekt[#x].hmiTrybAutoManual = 1 THEN
	                    IF #obiekt[#x].outStartUrządzenie = 0 THEN
	                        #obiekt[#x].hmiStanUrządzenia := 2;
	                    END_IF;
	                    IF #obiekt[#x].outStartUrządzenie = 1 THEN
	                        #obiekt[#x].hmiStanUrządzenia := 4;
	                    END_IF;
	                    IF #obiekt[#x].Awaria = 1 THEN
	                        #obiekt[#x].hmiStanUrządzenia := 6;
	                    END_IF;
	                END_IF;
	            END_REGION
	        5:  // Termometr
	            REGION typ5
	                
	                
	                //skalowanie
	                #obiekt[#x].kodBłedu := SCALE(IN := #obiekt[#x].inPomiarRaw,
	                                              HI_LIM := #obiekt[#x].maxskali,
	                                              LO_LIM := #obiekt[#x].minSkali,
	                                              BIPOLAR := 0,
	                                              OUT => #obiekt[#x].pomiarTymczas);
	                
	                //filtrowanie
	                #obiekt[#x].wyjTymczas := (#obiekt[#x].pomiarTymczas * (1 - #obiekt[#x].tFiltr)) + (#obiekt[#x].tFiltr * #obiekt[#x].WartośćPomiaru);
	                #obiekt[#x].WartośćPomiaru := #obiekt[#x].wyjTymczas;
	                
	                //symulacja
	                IF #obiekt[#x].hmiSymulujSygnałyWejsciowe THEN
	                    #obiekt[#x].WartośćPomiaru := #obiekt[#x].hmiSymulowanaWartośćAnalogowa;
	                    IF #obiekt[#x].hmiSymulowanaWartośćAnalogowa < #obiekt[#x].minSkali THEN
	                        #obiekt[#x].hmiSymulowanaWartośćAnalogowa := #obiekt[#x].minSkali;
	                    END_IF;
	                    IF #obiekt[#x].hmiSymulowanaWartośćAnalogowa > #obiekt[#x].maxskali THEN
	                        #obiekt[#x].hmiSymulowanaWartośćAnalogowa := #obiekt[#x].maxskali;
	                    END_IF;
	                END_IF;
	                //wyrzucanie bledu pomiaru
	                IF (#obiekt[#x].kodBłedu <> 0) AND (#obiekt[#x].czasDoAwariiPV < 10000) THEN
	                    
	                    #obiekt[#x].czasDoAwariiPV := #obiekt[#x].czasDoAwariiPV + 1;
	                    
	                    IF #obiekt[#x].czasDoAwariiPV > #obiekt[#x].czasDoAwariiSP THEN
	                        #obiekt[#x].Awaria := 1;
	                    END_IF;
	                    
	                ELSE
	                    #obiekt[#x].Awaria := 0;
	                    #obiekt[#x].czasDoAwariiPV := 0;
	                END_IF;
	                
	            END_REGION
	        6,18: //Ciśnieniomierz  
	            REGION typ6
	                
	                
	                
	                //skalowanie
	                #obiekt[#x].kodBłedu := SCALE(IN := #obiekt[#x].inPomiarRaw,
	                                              HI_LIM := #obiekt[#x].maxskali,
	                                              LO_LIM := #obiekt[#x].minSkali,
	                                              BIPOLAR := 0,
	                                              OUT => #obiekt[#x].pomiarTymczas);
	                
	                //filtrowanie
	                #obiekt[#x].wyjTymczas := (#obiekt[#x].pomiarTymczas * (1 - #obiekt[#x].tFiltr)) + (#obiekt[#x].tFiltr * #obiekt[#x].WartośćPomiaru);
	                #obiekt[#x].WartośćPomiaru := #obiekt[#x].wyjTymczas;
	                
	                //symulacja
	                IF #obiekt[#x].hmiSymulujSygnałyWejsciowe THEN
	                    #obiekt[#x].WartośćPomiaru := #obiekt[#x].hmiSymulowanaWartośćAnalogowa;
	                    IF #obiekt[#x].hmiSymulowanaWartośćAnalogowa < #obiekt[#x].minSkali THEN
	                        #obiekt[#x].hmiSymulowanaWartośćAnalogowa := #obiekt[#x].minSkali;
	                    END_IF;
	                    IF #obiekt[#x].hmiSymulowanaWartośćAnalogowa > #obiekt[#x].maxskali THEN
	                        #obiekt[#x].hmiSymulowanaWartośćAnalogowa := #obiekt[#x].maxskali;
	                    END_IF;
	                END_IF;
	                //wyrzucanie bledu pomiaru
	                IF (#obiekt[#x].kodBłedu <> 0) AND (#obiekt[#x].czasDoAwariiPV < 10000) THEN
	                    
	                    #obiekt[#x].czasDoAwariiPV := #obiekt[#x].czasDoAwariiPV + 1;
	                    
	                    IF #obiekt[#x].czasDoAwariiPV > #obiekt[#x].czasDoAwariiSP THEN
	                        #obiekt[#x].Awaria := 1;
	                    END_IF;
	                    
	                ELSE
	                    #obiekt[#x].Awaria := 0;
	                    #obiekt[#x].czasDoAwariiPV := 0;
	                END_IF;
	            END_REGION
	            
	            
	            
	        12: //CT stęzenie
	            REGION typ12
	                
	                
	                
	                //skalowanie
	                #obiekt[#x].kodBłedu := SCALE(IN := #obiekt[#x].inPomiarRaw,
	                                              HI_LIM := #obiekt[#x].maxskali,
	                                              LO_LIM := #obiekt[#x].minSkali,
	                                              BIPOLAR := 0,
	                                              OUT => #obiekt[#x].pomiarTymczas);
	                
	                //filtrowanie
	                #obiekt[#x].wyjTymczas := (#obiekt[#x].pomiarTymczas * (1 - #obiekt[#x].tFiltr))
	                + (#obiekt[#x].tFiltr * #obiekt[#x].pid_Rampa);
	                #obiekt[#x].pid_Rampa := #obiekt[#x].wyjTymczas;
	                #obiekt[#x].WartośćPomiaru := #obiekt[#x].wyjTymczas;
	                
	                //symulacja
	                IF #obiekt[#x].hmiSymulujSygnałyWejsciowe THEN
	                    #obiekt[#x].WartośćPomiaru := #obiekt[#x].hmiSymulowanaWartośćAnalogowa;
	                    IF #obiekt[#x].hmiSymulowanaWartośćAnalogowa < #obiekt[#x].minSkali THEN
	                        #obiekt[#x].hmiSymulowanaWartośćAnalogowa := #obiekt[#x].minSkali;
	                    END_IF;
	                    IF #obiekt[#x].hmiSymulowanaWartośćAnalogowa > #obiekt[#x].maxskali THEN
	                        #obiekt[#x].hmiSymulowanaWartośćAnalogowa := #obiekt[#x].maxskali;
	                    END_IF;
	                END_IF;
	                //wyrzucanie bledu pomiaru
	                IF (#obiekt[#x].kodBłedu <> 0) AND (#obiekt[#x].czasDoAwariiPV < 10000) THEN
	                    
	                    #obiekt[#x].czasDoAwariiPV := #obiekt[#x].czasDoAwariiPV + 1;
	                    
	                    IF #obiekt[#x].czasDoAwariiPV > #obiekt[#x].czasDoAwariiSP THEN
	                        #obiekt[#x].Awaria := 1;
	                    END_IF;
	                    
	                ELSE
	                    #obiekt[#x].Awaria := 0;
	                    #obiekt[#x].czasDoAwariiPV := 0;
	                END_IF;
	            END_REGION
	            
	            
	            
	            
	            
	        7: //Przepływomierz 
	            REGION typ7
	                
	                
	                
	                
	                //skalowanie
	                #obiekt[#x].kodBłedu := SCALE(IN := #obiekt[#x].inPomiarRaw,
	                                              HI_LIM := #obiekt[#x].maxskali,
	                                              LO_LIM := #obiekt[#x].minSkali,
	                                              BIPOLAR := 0,
	                                              OUT => #obiekt[#x].pomiarTymczas);
	                #obiekt[#x].hmiMetry3NaImpuls := #obiekt[#x].pomiarTymczas / 36000.0;// ile litrow co 100ms leci w rurze
	                //filtrowanie
	                //
	                #obiekt[#x].tFiltr := 0.9;
	                #obiekt[#x].wyjTymczas := (#obiekt[#x].pomiarTymczas *
	                (1 - #obiekt[#x].tFiltr)) + (#obiekt[#x].tFiltr * #obiekt[#x].WartośćPomiaru);
	                #obiekt[#x].WartośćPomiaru := #obiekt[#x].wyjTymczas;
	                
	                //symulacja
	                IF #obiekt[#x].hmiSymulujSygnałyWejsciowe THEN
	                    #obiekt[#x].WartośćPomiaru := #obiekt[#x].hmiSymulowanaWartośćAnalogowa;
	                    IF #obiekt[#x].hmiSymulowanaWartośćAnalogowa < #obiekt[#x].minSkali THEN
	                        #obiekt[#x].hmiSymulowanaWartośćAnalogowa := #obiekt[#x].minSkali;
	                    END_IF;
	                    IF #obiekt[#x].hmiSymulowanaWartośćAnalogowa > #obiekt[#x].maxskali THEN
	                        #obiekt[#x].hmiSymulowanaWartośćAnalogowa := #obiekt[#x].maxskali;
	                    END_IF;
	                END_IF;
	                //wyrzucanie bledu pomiaru
	                IF (#obiekt[#x].kodBłedu <> 0) AND (#obiekt[#x].czasDoAwariiPV < 10000) THEN
	                    
	                    #obiekt[#x].czasDoAwariiPV := #obiekt[#x].czasDoAwariiPV + 1;
	                    
	                    IF #obiekt[#x].czasDoAwariiPV > #obiekt[#x].czasDoAwariiSP THEN
	                        #obiekt[#x].Awaria := 1;
	                    END_IF;
	                    
	                ELSE
	                    #obiekt[#x].Awaria := 0;
	                    #obiekt[#x].czasDoAwariiPV := 0;
	                END_IF;
	                
	                
	                // //licznikimpulsów i metrów sześciennych
	                // //symulacja
	                // IF #obiekt[#x].hmiSymulujSygnałyWejsciowe THEN
	                //     #obiekt[#x].licznikTotalImpulsy := #obiekt[#x].licznikTotalImpulsy + 1;
	                //     IF #obiekt[#x].licznikTotalImpulsy > 1000.0 / #obiekt[#x].hmiSymulowanaWartośćAnalogowa / 2.0 THEN
	                //         #obiekt[#x].diImpulsy := 1;
	                //     END_IF;
	                //     IF #obiekt[#x].licznikTotalImpulsy > 1000.0 / #obiekt[#x].hmiSymulowanaWartośćAnalogowa THEN
	                //         #obiekt[#x].licznikTotalImpulsy := 0;
	                //         #obiekt[#x].diImpulsy := 0;
	                //     END_IF;
	                // END_IF;
	                
	                // //zliczanie litrow po impulsach
	                
	                // IF #obiekt[#x].diImpulsy AND NOT #obiekt[#x].R_Trig THEN // warunek spełniony przy zboczu narastającym
	                
	                //     IF #obiekt[#x].startLicznik1 THEN
	                //         #obiekt[#x].licznik1 := #obiekt[#x].licznik1 + #obiekt[#x].hmiMetry3NaImpuls;
	                //     END_IF;
	                //     IF #obiekt[#x].startLicznik2 THEN
	                //         #obiekt[#x].licznik2 := #obiekt[#x].licznik2 + #obiekt[#x].hmiMetry3NaImpuls;
	                //     END_IF;
	                //     IF #obiekt[#x].startLicznik3 THEN
	                //         #obiekt[#x].licznik3 := #obiekt[#x].licznik3 + #obiekt[#x].hmiMetry3NaImpuls;
	                //     END_IF;
	                
	                // END_IF;
	                // #obiekt[#x].R_Trig := #obiekt[#x].diImpulsy;
	                
	                //zliczanie litrow po impulsach
	                
	                ////nowe zliczanie po wartosci co 100mS
	                //
	                IF #obiekt[#x].hmiSymulujSygnałyWejsciowe THEN
	                    #obiekt[#x].WartośćPomiaru := #obiekt[#x].hmiSymulowanaWartośćAnalogowa;
	                    #obiekt[#x].hmiMetry3NaImpuls := #obiekt[#x].hmiSymulowanaWartośćAnalogowa / 36000.0;
	                END_IF;
	                
	                
	                IF #obiekt[#x].startLicznik1 THEN
	                    #obiekt[#x].licznik1 := #obiekt[#x].licznik1 + #obiekt[#x].hmiMetry3NaImpuls;
	                END_IF;
	                
	                
	                IF #obiekt[#x].startLicznik2 THEN
	                    #obiekt[#x].licznik2 := #obiekt[#x].licznik2 + #obiekt[#x].hmiMetry3NaImpuls;
	                END_IF;
	                IF #obiekt[#x].startLicznik3 THEN
	                    #obiekt[#x].licznik3 := #obiekt[#x].licznik3 + #obiekt[#x].hmiMetry3NaImpuls;
	                END_IF;
	                
	                //takie tam zeby diodka impulsowala
	                //
	                #obiekt[#x].diImpulsy := #obiekt[#x].diImpulsy;
	                
	                ////////
	                
	                
	                
	                
	                
	                #obiekt[#x].R_Trig := #obiekt[#x].diImpulsy;
	                
	                // kasowanie liczników
	                IF #obiekt[#x].zerujLicznik1 THEN
	                    #obiekt[#x].licznik1 := 0.0;
	                END_IF;
	                IF #obiekt[#x].zerujLicznik2 THEN
	                    #obiekt[#x].licznik2 := 0.0;
	                END_IF;
	                IF #obiekt[#x].zerujLicznik3 THEN
	                    #obiekt[#x].licznik3 := 0.0;
	                END_IF;
	            END_REGION
	        8://PID
	            REGION typ8
	                
	                
	                ;
	                IF #obiekt[#x].inZadaneWysterowanieAuto = 0.0 THEN
	                    #obiekt[#x].hmiStanUrządzenia := 0;
	                END_IF;
	                IF #obiekt[#x].inZadaneWysterowanieAuto <> 0.0 THEN
	                    #obiekt[#x].hmiStanUrządzenia := 1;
	                END_IF;
	                IF #obiekt[#x].hmiTrybAutoManual THEN
	                    #obiekt[#x].hmiStanUrządzenia := 2;
	                END_IF;
	            END_REGION
	        9: //czujnik cyfrowy ONOFF
	            REGION typ9
	                
	                
	                // stan urządzenia DO stacyjki
	                IF #obiekt[#x].hmiPotwWysterowania THEN
	                    #obiekt[#x].hmiStanUrządzenia := 3;
	                ELSE
	                    #obiekt[#x].hmiStanUrządzenia := 1;
	                END_IF;
	                // stan urządzenia DO stacyjki w symulacji
	                IF #obiekt[#x].hmiSymulujSygnałyWejsciowe THEN
	                    #obiekt[#x].hmiPotwWysterowania := #obiekt[#x].hmiSymulacjaPotwWysterowania;
	                    IF #obiekt[#x].hmiPotwWysterowania THEN
	                        #obiekt[#x].hmiStanUrządzenia := 4;
	                    ELSE
	                        #obiekt[#x].hmiStanUrządzenia := 2;
	                    END_IF;
	                ELSE
	                    
